C05459=1073.905,147.955,426.139,173.670,25.621,154.541
C05460=1073.899,147.705,426.161,173.668,25.618,154.541
C05461=1073.894,147.456,426.181,173.666,25.616,154.541
C05462=1073.888,147.208,426.202,173.664,25.613,154.541
C05463=1073.882,146.958,426.223,173.663,25.610,154.540
C05464=1073.877,146.709,426.244,173.661,25.608,154.540
C05465=1073.871,146.461,426.265,173.659,25.606,154.540
C05466=1073.865,146.211,426.286,173.657,25.603,154.539
C05467=1073.859,145.962,426.306,173.655,25.600,154.539
C05468=1073.854,145.714,426.327,173.654,25.598,154.539
C05469=1073.848,145.464,426.348,173.651,25.595,154.538
C05470=1073.843,145.215,426.369,173.650,25.592,154.538
C05471=1073.837,144.966,426.390,173.647,25.590,154.538
C05472=1073.830,144.717,426.410,173.646,25.587,154.537
C05473=1073.825,144.467,426.431,173.645,25.585,154.537
C05474=1073.820,144.219,426.452,173.642,25.582,154.537
C05475=1073.814,143.970,426.472,173.641,25.580,154.537
C05476=1073.808,143.720,426.493,173.638,25.577,154.536
C05477=1073.802,143.438,426.517,173.637,25.574,154.536
C05478=1073.795,143.157,426.540,173.635,25.571,154.535
C05479=1073.789,142.875,426.564,173.633,25.568,154.535
C05480=1073.782,142.593,426.586,173.630,25.565,154.535
C05481=1073.777,142.344,426.608,173.629,25.562,154.534
C05482=1073.771,142.094,426.628,173.626,25.560,154.534
C05483=1073.766,141.845,426.649,173.625,25.558,154.534
C05484=1073.760,141.596,426.669,173.624,25.555,154.533
C05485=1073.755,141.347,426.690,173.621,25.552,154.533
C05486=1073.748,141.098,426.711,173.620,25.550,154.533
C05487=1073.742,140.849,426.731,173.618,25.547,154.533
C05488=1073.737,140.600,426.752,173.616,25.544,154.532
C05489=1073.732,140.351,426.772,173.615,25.542,154.532
C05490=1073.727,140.102,426.793,173.612,25.539,154.532
C05491=1073.720,139.852,426.813,173.611,25.537,154.531
C05492=1073.715,139.603,426.834,173.609,25.534,154.531
C05493=1073.708,139.355,426.854,173.607,25.531,154.531
C05494=1073.703,139.106,426.875,173.606,25.529,154.530
C05495=1073.697,138.856,426.896,173.603,25.526,154.530
C05496=1073.691,138.607,426.916,173.602,25.523,154.530
C05497=1073.686,138.358,426.936,173.600,25.521,154.529
C05498=1073.680,138.109,426.956,173.598,25.518,154.529
C05499=1073.675,137.860,426.977,173.597,25.516,154.529
C05500=1073.668,137.611,426.997,173.595,25.513,154.528
C05501=1073.663,137.362,427.018,173.593,25.511,154.528
C05502=1073.658,137.112,427.038,173.591,25.508,154.528
C05503=1073.652,136.864,427.058,173.589,25.505,154.527
C05504=1073.647,136.615,427.079,173.588,25.503,154.527
C05505=1073.641,136.366,427.099,173.586,25.500,154.527
C05506=1073.635,136.116,427.120,173.584,25.497,154.527
C05507=1073.629,135.867,427.140,173.582,25.495,154.526
C05508=1073.623,135.618,427.160,173.580,25.493,154.526
C05509=1073.617,135.369,427.180,173.579,25.490,154.526
C05510=1073.612,135.120,427.201,173.577,25.487,154.525
C05511=1073.606,134.871,427.221,173.575,25.485,154.525
C05512=1073.600,134.621,427.242,173.574,25.482,154.525
C05513=1073.594,134.373,427.262,173.572,25.479,154.524
C05514=1073.589,134.123,427.282,173.570,25.477,154.524
C05515=1073.583,133.875,427.302,173.568,25.474,154.524
C05516=1073.578,133.625,427.322,173.566,25.472,154.523
C05517=1073.572,133.376,427.342,173.565,25.469,154.523
C05518=1073.567,133.127,427.362,173.563,25.466,154.523
C05519=1073.561,132.878,427.382,173.561,25.464,154.522
C05520=1073.555,132.628,427.403,173.560,25.461,154.522
C05521=1073.549,132.379,427.423,173.558,25.458,154.522
C05522=1073.544,132.130,427.444,173.556,25.456,154.522
C05523=1073.538,131.881,427.463,173.555,25.454,154.521
C05524=1073.532,131.632,427.483,173.552,25.450,154.521
C05525=1073.527,131.383,427.504,173.551,25.448,154.521
C05526=1073.521,131.134,427.523,173.549,25.446,154.520
C05527=1073.515,130.885,427.543,173.547,25.443,154.520
C05528=1073.509,130.635,427.563,173.546,25.440,154.520
C05529=1073.503,130.386,427.584,173.544,25.438,154.519
C05530=1073.497,130.137,427.604,173.542,25.435,154.519
C05531=1073.491,129.888,427.624,173.541,25.433,154.519
C05532=1073.486,129.639,427.643,173.538,25.430,154.518
C05533=1073.480,129.390,427.663,173.537,25.428,154.518
C05534=1073.474,129.141,427.683,173.535,25.425,154.518
C05535=1073.468,128.892,427.703,173.533,25.423,154.518
C05536=1073.462,128.642,427.723,173.532,25.420,154.517
C05537=1073.456,128.393,427.743,173.530,25.418,154.517
C05538=1073.451,128.144,427.763,173.528,25.415,154.517
C05539=1073.445,127.895,427.783,173.527,25.413,154.516
C05540=1073.439,127.646,427.803,173.525,25.410,154.516
C05541=1073.431,127.300,427.830,173.522,25.406,154.516
C05542=1073.423,126.955,427.858,173.520,25.403,154.515
C05543=1073.416,126.610,427.885,173.518,25.399,154.515
C05544=1073.407,126.264,427.912,173.516,25.396,154.514
C05545=1073.402,126.047,427.930,173.514,25.393,154.514
C05546=1073.398,125.829,427.947,173.513,25.391,154.514
C05547=1073.392,125.612,427.965,173.510,25.388,154.513
C05548=1073.387,125.394,427.981,173.509,25.386,154.513
C05549=1073.382,125.177,427.999,173.507,25.384,154.513
C05550=1073.377,124.959,428.017,173.506,25.382,154.513
C05551=1073.372,124.742,428.034,173.504,25.380,154.512
C05552=1073.367,124.524,428.051,173.503,25.377,154.512
C05553=1073.361,124.276,428.071,173.502,25.375,154.512
C05554=1073.355,124.026,428.090,173.500,25.372,154.511
C05555=1073.349,123.777,428.110,173.498,25.370,154.511
C05556=1073.344,123.528,428.130,173.497,25.367,154.511
C05557=1073.338,123.279,428.150,173.495,25.364,154.510
C05558=1073.333,123.029,428.169,173.493,25.362,154.510
C05559=1073.327,122.781,428.189,173.491,25.359,154.510
C05560=1073.321,122.531,428.208,173.490,25.357,154.509
C05561=1073.315,122.282,428.228,173.488,25.353,154.509
C05562=1073.310,122.033,428.248,173.486,25.351,154.509
C05563=1073.304,121.784,428.268,173.485,25.349,154.508
C05564=1073.298,121.534,428.287,173.484,25.346,154.508
C05565=1073.293,121.285,428.306,173.481,25.343,154.508
C05566=1073.287,121.037,428.326,173.480,25.341,154.508
C05567=1073.282,120.787,428.345,173.478,25.338,154.507
C05568=1073.276,120.538,428.365,173.476,25.336,154.507
C05569=1073.271,120.289,428.385,173.475,25.333,154.506
C05570=1073.265,120.039,428.404,173.473,25.330,154.506
C05571=1073.259,119.791,428.424,173.471,25.328,154.506
C05572=1073.253,119.541,428.444,173.470,25.325,154.506
C05573=1073.247,119.292,428.463,173.468,25.323,154.505
C05574=1073.242,119.043,428.483,173.467,25.320,154.505
C05575=1073.236,118.793,428.502,173.465,25.317,154.505
C05576=1073.230,118.545,428.522,173.463,25.314,154.504
C05577=1073.225,118.296,428.541,173.462,25.312,154.504
C05578=1073.220,118.046,428.561,173.459,25.309,154.504
C05579=1073.214,117.797,428.581,173.458,25.306,154.503
C05580=1073.208,117.548,428.600,173.457,25.304,154.503
C05581=1073.203,117.298,428.619,173.454,25.301,154.503
C05582=1073.197,117.050,428.639,173.453,25.299,154.502
C05583=1073.191,116.800,428.658,173.452,25.296,154.502
C05584=1073.185,116.551,428.678,173.450,25.293,154.502
C05585=1073.180,116.302,428.696,173.448,25.290,154.501
C05586=1073.174,116.053,428.716,173.447,25.288,154.501
C05587=1073.168,115.804,428.736,173.445,25.285,154.500
C05588=1073.163,115.554,428.755,173.443,25.282,154.500
C05589=1073.157,115.305,428.774,173.442,25.280,154.500
C05590=1073.152,115.057,428.794,173.440,25.277,154.500
C05591=1073.146,114.807,428.813,173.439,25.275,154.499
C05592=1073.141,114.558,428.833,173.437,25.272,154.499
C05593=1073.135,114.308,428.852,173.435,25.269,154.499
C05594=1073.129,114.059,428.871,173.434,25.267,154.498
C05595=1073.123,113.810,428.891,173.432,25.264,154.498
C05596=1073.117,113.561,428.910,173.430,25.261,154.497
C05597=1073.112,113.312,428.929,173.429,25.259,154.497
C05598=1073.107,113.063,428.948,173.427,25.256,154.497
C05599=1073.101,112.813,428.967,173.425,25.253,154.497
C05600=1073.095,112.564,428.986,173.424,25.251,154.496
C05601=1073.089,112.314,429.006,173.422,25.248,154.496
C05602=1073.083,112.065,429.024,173.421,25.246,154.496
C05603=1073.078,111.817,429.044,173.419,25.243,154.495
C05604=1073.072,111.568,429.063,173.417,25.240,154.495
C05605=1073.065,111.285,429.085,173.416,25.237,154.494
C05606=1073.058,111.003,429.107,173.414,25.235,154.494
C05607=1073.052,110.721,429.128,173.411,25.232,154.494
C05608=1073.045,110.439,429.149,173.410,25.229,154.493
C05609=1073.040,110.189,429.168,173.409,25.226,154.493
C05610=1073.035,109.940,429.187,173.406,25.223,154.493
C05611=1073.029,109.692,429.207,173.405,25.221,154.493
C05612=1073.022,109.442,429.226,173.404,25.219,154.492
C05613=1073.017,109.193,429.245,173.402,25.216,154.492
C05614=1073.011,108.944,429.264,173.400,25.213,154.492
C05615=1073.004,108.694,429.283,173.399,25.210,154.491
C05616=1073.000,108.445,429.301,173.397,25.208,154.491
C05617=1072.994,108.196,429.320,173.396,25.205,154.491
C05618=1072.988,107.947,429.339,173.394,25.202,154.490
C05619=1072.982,107.697,429.358,173.392,25.200,154.490
C05620=1072.977,107.448,429.377,173.391,25.197,154.489
C05621=1072.971,107.199,429.396,173.389,25.195,154.489
C05622=1072.965,106.950,429.415,173.387,25.192,154.489
C05623=1072.959,106.700,429.434,173.386,25.189,154.489
C05624=1072.953,106.451,429.453,173.384,25.187,154.488
C05625=1072.948,106.203,429.472,173.383,25.184,154.488
C05626=1072.942,105.953,429.491,173.381,25.181,154.488
C05627=1072.936,105.704,429.510,173.379,25.179,154.487
C05628=1072.930,105.455,429.528,173.378,25.176,154.487
C05629=1072.925,105.205,429.547,173.377,25.174,154.487
C05630=1072.919,104.956,429.566,173.374,25.171,154.486
C05631=1072.913,104.707,429.585,173.373,25.168,154.486
C05632=1072.908,104.458,429.604,173.372,25.166,154.486
C05633=1072.902,104.208,429.623,173.370,25.163,154.485
C05634=1072.896,103.959,429.642,173.368,25.160,154.485
C05635=1072.891,103.710,429.660,173.367,25.158,154.485
C05636=1072.885,103.461,429.679,173.365,25.155,154.484
C05637=1072.879,103.211,429.698,173.364,25.152,154.484
C05638=1072.873,102.962,429.717,173.361,25.150,154.484
C05639=1072.867,102.714,429.735,173.360,25.147,154.483
C05640=1072.862,102.464,429.754,173.359,25.145,154.483
C05641=1072.856,102.214,429.773,173.357,25.142,154.483
C05642=1072.850,101.966,429.791,173.356,25.139,154.482
C05643=1072.845,101.716,429.811,173.354,25.136,154.482
C05644=1072.839,101.466,429.829,173.352,25.134,154.482
C05645=1072.833,101.218,429.847,173.351,25.131,154.481
C05646=1072.828,100.968,429.867,173.350,25.129,154.481
C05647=1072.821,100.719,429.885,173.347,25.125,154.481
C05648=1072.817,100.470,429.903,173.346,25.123,154.480
C05649=1072.810,100.221,429.922,173.345,25.121,154.480
C05650=1072.804,99.971,429.941,173.343,25.118,154.480
C05651=1072.799,99.722,429.959,173.342,25.116,154.479
C05652=1072.792,99.473,429.977,173.340,25.113,154.479
C05653=1072.787,99.224,429.997,173.338,25.110,154.479
C05654=1072.781,98.975,430.014,173.337,25.108,154.478
C05655=1072.776,98.725,430.034,173.336,25.105,154.478
C05656=1072.769,98.476,430.052,173.333,25.102,154.478
C05657=1072.764,98.227,430.070,173.332,25.099,154.477
C05658=1072.758,97.978,430.089,173.331,25.097,154.477
C05659=1072.752,97.728,430.107,173.329,25.095,154.477
C05660=1072.747,97.479,430.126,173.328,25.092,154.476
C05661=1072.740,97.230,430.144,173.325,25.089,154.476
C05662=1072.734,96.980,430.162,173.324,25.086,154.476
C05663=1072.729,96.732,430.181,173.323,25.084,154.475
C05664=1072.723,96.482,430.199,173.321,25.081,154.475
C05665=1072.717,96.232,430.218,173.320,25.079,154.475
C05666=1072.712,95.983,430.236,173.318,25.076,154.474
C05667=1072.705,95.734,430.255,173.316,25.073,154.474
C05668=1072.701,95.485,430.273,173.315,25.071,154.474
C05669=1072.693,95.203,430.294,173.313,25.068,154.473
C05670=1072.687,94.921,430.315,173.312,25.065,154.473
C05671=1072.681,94.639,430.336,173.309,25.062,154.473
C05672=1072.674,94.356,430.356,173.308,25.059,154.472
C05673=1072.669,94.107,430.375,173.307,25.056,154.472
C05674=1072.662,93.858,430.393,173.305,25.054,154.471
C05675=1072.657,93.609,430.411,173.303,25.051,154.471
C05676=1072.651,93.360,430.430,173.302,25.048,154.471
C05677=1072.646,93.110,430.448,173.300,25.046,154.470
C05678=1072.639,92.861,430.466,173.299,25.043,154.470
C05679=1072.634,92.611,430.485,173.298,25.040,154.470
C05680=1072.628,92.363,430.503,173.295,25.037,154.469
C05681=1072.622,92.113,430.521,173.294,25.035,154.469
C05682=1072.617,91.864,430.539,173.293,25.032,154.469
C05683=1072.611,91.615,430.558,173.291,25.030,154.468
C05684=1072.605,91.366,430.575,173.290,25.027,154.468
C05685=1072.599,91.116,430.595,173.288,25.024,154.468
C05686=1072.594,90.867,430.612,173.286,25.021,154.467
C05687=1072.588,90.617,430.630,173.285,25.019,154.467
C05688=1072.582,90.369,430.648,173.284,25.016,154.467
C05689=1072.577,90.119,430.667,173.282,25.014,154.466
C05690=1072.570,89.869,430.685,173.280,25.010,154.466
C05691=1072.565,89.621,430.703,173.279,25.008,154.466
C05692=1072.559,89.371,430.721,173.277,25.006,154.465
C05693=1072.553,89.122,430.739,173.276,25.003,154.465
C05694=1072.547,88.873,430.757,173.275,25.001,154.465
C05695=1072.541,88.624,430.775,173.272,24.997,154.464
C05696=1072.535,88.374,430.793,173.271,24.995,154.464
C05697=1072.530,88.125,430.811,173.270,24.993,154.464
C05698=1072.524,87.876,430.830,173.268,24.990,154.463
C05699=1072.518,87.627,430.847,173.267,24.987,154.463
C05700=1072.512,87.377,430.865,173.266,24.985,154.463
C05701=1072.507,87.128,430.883,173.263,24.982,154.462
C05702=1072.500,86.879,430.901,173.262,24.979,154.462
C05703=1072.495,86.630,430.919,173.261,24.977,154.462
C05704=1072.489,86.380,430.937,173.259,24.974,154.461
C05705=1072.483,86.131,430.954,173.258,24.971,154.461
C05706=1072.477,85.881,430.972,173.256,24.969,154.461
C05707=1072.472,85.632,430.991,173.254,24.966,154.460
C05708=1072.466,85.383,431.009,173.253,24.964,154.460
C05709=1072.460,85.134,431.027,173.252,24.961,154.460
C05710=1072.454,84.884,431.045,173.250,24.958,154.459
C05711=1072.448,84.635,431.062,173.249,24.955,154.459
C05712=1072.442,84.386,431.081,173.247,24.953,154.459
C05713=1072.437,84.137,431.098,173.245,24.950,154.458
C05714=1072.430,83.887,431.116,173.244,24.948,154.458
C05715=1072.425,83.638,431.134,173.243,24.945,154.458
C05716=1072.419,83.388,431.152,173.241,24.942,154.457
C05717=1072.413,83.139,431.169,173.240,24.939,154.457
C05718=1072.408,82.890,431.187,173.238,24.937,154.457
C05719=1072.402,82.640,431.205,173.236,24.934,154.456
C05720=1072.396,82.391,431.222,173.235,24.932,154.456
C05721=1072.390,82.142,431.240,173.234,24.929,154.456
C05722=1072.385,81.893,431.259,173.232,24.926,154.455
C05723=1072.379,81.643,431.277,173.231,24.923,154.455
C05724=1072.373,81.394,431.295,173.229,24.921,154.455
C05725=1072.368,81.145,431.312,173.227,24.918,154.454
C05726=1072.362,80.895,431.330,173.226,24.916,154.454
C05727=1072.356,80.646,431.348,173.225,24.913,154.454
C05728=1072.350,80.396,431.366,173.223,24.910,154.453
C05729=1072.344,80.147,431.383,173.222,24.907,154.453
C05730=1072.339,79.898,431.401,173.220,24.905,154.453
C05731=1072.333,79.649,431.419,173.218,24.902,154.452
C05732=1072.327,79.400,431.436,173.217,24.900,154.452
C05733=1072.321,79.117,431.456,173.216,24.897,154.452
C05734=1072.314,78.835,431.476,173.214,24.893,154.451
C05735=1072.307,78.554,431.496,173.212,24.891,154.451
C05736=1072.301,78.271,431.516,173.210,24.887,154.450
C05737=1072.295,78.022,431.533,173.209,24.884,154.450
C05738=1072.289,77.773,431.551,173.207,24.882,154.450
C05739=1072.284,77.524,431.569,173.206,24.879,154.449
C05740=1072.278,77.274,431.586,173.205,24.877,154.449
C05741=1072.271,77.025,431.604,173.203,24.874,154.449
C05742=1072.266,76.776,431.621,173.201,24.871,154.448
C05743=1072.260,76.526,431.639,173.200,24.868,154.448
C05744=1072.255,76.277,431.656,173.198,24.866,154.448
C05745=1072.249,76.028,431.674,173.197,24.863,154.447
C05746=1072.242,75.778,431.691,173.196,24.861,154.447
C05747=1072.237,75.529,431.709,173.194,24.858,154.447
C05748=1072.231,75.280,431.726,173.193,24.856,154.446
C05749=1072.225,75.030,431.744,173.191,24.853,154.446
C05750=1072.220,74.781,431.761,173.190,24.850,154.446
C05751=1072.214,74.532,431.778,173.188,24.848,154.445
C05752=1072.207,74.282,431.796,173.187,24.845,154.445
C05753=1072.202,74.033,431.813,173.185,24.842,154.445
C05754=1072.196,73.784,431.831,173.184,24.840,154.444
C05755=1072.191,73.534,431.848,173.183,24.837,154.444
C05756=1072.184,73.285,431.865,173.181,24.834,154.444
C05757=1072.179,73.036,431.883,173.179,24.832,154.443
C05758=1072.173,72.786,431.901,173.178,24.829,154.443
C05759=1072.167,72.537,431.918,173.177,24.826,154.443
C05760=1072.161,72.288,431.935,173.175,24.823,154.442
C05761=1072.155,72.038,431.952,173.174,24.821,154.442
C05762=1072.150,71.789,431.970,173.173,24.818,154.441
C05763=1072.144,71.539,431.987,173.170,24.816,154.441
C05764=1072.138,71.291,432.004,173.169,24.813,154.441
C05765=1072.132,71.041,432.022,173.168,24.810,154.441
C05766=1072.126,70.792,432.039,173.166,24.807,154.440
C05767=1072.121,70.542,432.056,173.165,24.805,154.440
C05768=1072.114,70.293,432.074,173.164,24.802,154.439
C05769=1072.109,70.044,432.091,173.162,24.800,154.439
C05770=1072.104,69.794,432.108,173.160,24.797,154.439
C05771=1072.097,69.545,432.125,173.159,24.794,154.439
C05772=1072.091,69.296,432.143,173.157,24.791,154.438
C05773=1072.086,69.046,432.160,173.156,24.789,154.438
C05774=1072.080,68.797,432.177,173.155,24.786,154.437
C05775=1072.075,68.548,432.194,173.153,24.784,154.437
C05776=1072.068,68.298,432.211,173.152,24.781,154.437
C05777=1072.062,68.049,432.228,173.150,24.778,154.436
C05778=1072.057,67.799,432.245,173.149,24.775,154.436
C05779=1072.051,67.551,432.262,173.147,24.773,154.436
C05780=1072.045,67.300,432.279,173.146,24.770,154.435
C05781=1072.039,67.052,432.296,173.145,24.768,154.435
C05782=1072.033,66.803,432.314,173.143,24.765,154.435
C05783=1072.028,66.553,432.331,173.142,24.762,154.434
C05784=1072.021,66.304,432.348,173.141,24.759,154.434
C05785=1072.016,66.054,432.365,173.138,24.757,154.434
C05786=1072.010,65.805,432.382,173.137,24.754,154.433
C05787=1072.004,65.555,432.399,173.136,24.752,154.433
C05788=1071.998,65.306,432.416,173.134,24.749,154.433
C05789=1071.992,65.056,432.433,173.133,24.746,154.432
C05790=1071.986,64.808,432.450,173.132,24.743,154.432
C05791=1071.981,64.558,432.467,173.130,24.741,154.432
C05792=1071.975,64.309,432.484,173.129,24.738,154.431
C05793=1071.969,64.059,432.501,173.127,24.735,154.431
C05794=1071.963,63.810,432.518,173.125,24.733,154.431
C05795=1071.957,63.561,432.534,173.124,24.730,154.430
C05796=1071.950,63.311,432.552,173.123,24.728,154.430
C05797=1071.944,63.029,432.570,173.121,24.725,154.430
C05798=1071.938,62.747,432.590,173.119,24.722,154.429
C05799=1071.930,62.465,432.609,173.118,24.719,154.429
C05800=1071.924,62.182,432.628,173.116,24.716,154.428
C05801=1071.918,61.934,432.645,173.115,24.713,154.428
C05802=1071.912,61.684,432.661,173.113,24.711,154.428
C05803=1071.906,61.434,432.678,173.112,24.708,154.428
C05804=1071.900,61.185,432.695,173.110,24.706,154.427
C05805=1071.894,60.936,432.712,173.109,24.703,154.427
C05806=1071.888,60.687,432.729,173.108,24.700,154.427
C05807=1071.882,60.437,432.745,173.106,24.698,154.426
C05808=1071.876,60.187,432.762,173.104,24.695,154.426
C05809=1071.870,59.939,432.779,173.103,24.692,154.426
C05810=1071.864,59.689,432.796,173.102,24.689,154.425
C05811=1071.858,59.440,432.812,173.100,24.687,154.425
C05812=1071.852,59.191,432.829,173.099,24.684,154.425
C05813=1071.846,58.940,432.846,173.098,24.682,154.424
C05814=1071.840,58.691,432.863,173.096,24.679,154.424
C05815=1071.834,58.442,432.879,173.095,24.677,154.424
C05816=1071.828,58.193,432.896,173.093,24.674,154.423
C05817=1071.823,57.943,432.913,173.091,24.671,154.423
C05818=1071.817,57.694,432.929,173.090,24.669,154.423
C05819=1071.811,57.445,432.945,173.089,24.666,154.422
C05820=1071.805,57.195,432.963,173.087,24.663,154.422
C05821=1071.799,56.946,432.979,173.086,24.660,154.422
C05822=1071.793,56.696,432.996,173.085,24.658,154.421
C05823=1071.787,56.447,433.012,173.083,24.655,154.421
C05824=1071.782,56.198,433.030,173.082,24.653,154.421
C05825=1071.776,55.949,433.046,173.080,24.650,154.420
C05826=1071.770,55.699,433.062,173.079,24.647,154.420
C05827=1071.764,55.450,433.078,173.077,24.645,154.420
C05828=1071.759,55.200,433.095,173.076,24.642,154.419
C05829=1071.752,54.951,433.112,173.075,24.640,154.419
C05830=1071.746,54.701,433.129,173.073,24.637,154.419
C05831=1071.740,54.452,433.145,173.072,24.634,154.418
C05832=1071.735,54.202,433.162,173.071,24.631,154.418
C05833=1071.729,53.953,433.178,173.069,24.629,154.418
C05834=1071.723,53.704,433.194,173.067,24.626,154.417
C05835=1071.716,53.455,433.211,173.066,24.623,154.417
C05836=1071.711,53.205,433.228,173.064,24.621,154.416
C05837=1071.705,52.956,433.244,173.063,24.618,154.416
C05838=1071.699,52.707,433.261,173.062,24.615,154.416
C05839=1071.693,52.457,433.277,173.060,24.613,154.416
C05840=1071.688,52.208,433.294,173.059,24.610,154.415
C05841=1071.682,51.958,433.310,173.058,24.608,154.415
C05842=1071.676,51.709,433.326,173.057,24.605,154.414
C05843=1071.670,51.460,433.343,173.055,24.602,154.414
C05844=1071.664,51.210,433.359,173.053,24.599,154.414
C05845=1071.659,50.961,433.376,173.052,24.597,154.413
C05846=1071.653,50.711,433.392,173.050,24.594,154.413
C05847=1071.647,50.462,433.408,173.049,24.591,154.413
C05848=1071.641,50.212,433.424,173.048,24.589,154.412
C05849=1071.635,49.964,433.441,173.046,24.586,154.412
C05850=1071.630,49.714,433.458,173.045,24.583,154.412
C05851=1071.624,49.465,433.475,173.044,24.581,154.411
C05852=1071.618,49.215,433.491,173.043,24.578,154.411
C05853=1071.612,48.966,433.507,173.041,24.576,154.411
C05854=1071.606,48.716,433.523,173.039,24.572,154.410
C05855=1071.601,48.466,433.539,173.038,24.570,154.410
C05856=1071.595,48.217,433.556,173.036,24.567,154.410
C05857=1071.589,47.968,433.572,173.035,24.565,154.409
C05858=1071.583,47.718,433.588,173.034,24.562,154.409
C05859=1071.577,47.469,433.604,173.032,24.559,154.409
C05860=1071.571,47.220,433.621,173.031,24.557,154.408
C05861=1071.565,46.937,433.640,173.029,24.553,154.408
C05862=1071.559,46.655,433.658,173.028,24.550,154.408
C05863=1071.552,46.372,433.676,173.027,24.547,154.407
C05864=1071.546,46.090,433.695,173.024,24.544,154.407
C05865=1071.540,45.840,433.711,173.023,24.541,154.406
C05866=1071.534,45.591,433.728,173.022,24.539,154.406
C05867=1071.528,45.342,433.743,173.021,24.536,154.406
C05868=1071.522,45.093,433.760,173.019,24.534,154.405
C05869=1071.517,44.843,433.775,173.018,24.531,154.405
C05870=1071.511,44.594,433.791,173.017,24.528,154.405
C05871=1071.506,44.344,433.808,173.015,24.525,154.404
C05872=1071.500,44.095,433.825,173.014,24.523,154.404
C05873=1071.494,43.845,433.841,173.012,24.520,154.404
C05874=1071.488,43.596,433.857,173.010,24.517,154.403
C05875=1071.482,43.346,433.873,173.009,24.515,154.403
C05876=1071.476,43.097,433.889,173.008,24.512,154.403
C05877=1071.470,42.847,433.905,173.007,24.509,154.402
C05878=1071.465,42.599,433.921,173.005,24.507,154.402
C05879=1071.458,42.350,433.937,173.004,24.504,154.402
C05880=1071.452,42.100,433.952,173.003,24.502,154.401
C05881=1071.447,41.850,433.969,173.001,24.499,154.401
C05882=1071.441,41.601,433.985,173.000,24.496,154.401
C05883=1071.435,41.352,434.001,172.999,24.493,154.400
C05884=1071.429,41.102,434.017,172.996,24.491,154.400
C05885=1071.423,40.852,434.033,172.995,24.488,154.400
C05886=1071.417,40.603,434.049,172.994,24.485,154.399
C05887=1071.411,40.353,434.065,172.992,24.483,154.399
C05888=1071.405,40.104,434.081,172.991,24.480,154.399
C05889=1071.400,39.855,434.097,172.990,24.478,154.398
C05890=1071.394,39.606,434.113,172.989,24.475,154.398
C05891=1071.389,39.356,434.129,172.987,24.472,154.398
C05892=1071.382,39.107,434.144,172.986,24.470,154.397
C05893=1071.376,38.857,434.160,172.985,24.467,154.397
C05894=1071.370,38.607,434.176,172.983,24.464,154.397
C05895=1071.364,38.358,434.192,172.982,24.462,154.396
C05896=1071.359,38.109,434.207,172.980,24.459,154.396
C05897=1071.353,37.859,434.224,172.978,24.456,154.396
C05898=1071.347,37.610,434.240,172.977,24.453,154.395
C05899=1071.341,37.360,434.255,172.976,24.451,154.395
C05900=1071.335,37.111,434.271,172.974,24.449,154.395
C05901=1071.329,36.862,434.287,172.973,24.446,154.394
C05902=1071.323,36.612,434.303,172.972,24.443,154.394
C05903=1071.317,36.363,434.319,172.971,24.440,154.394
C05904=1071.312,36.113,434.334,172.969,24.438,154.393
C05905=1071.306,35.864,434.350,172.968,24.436,154.393
C05906=1071.299,35.614,434.365,172.967,24.433,154.393
C05907=1071.293,35.365,434.381,172.964,24.430,154.392
C05908=1071.287,35.116,434.398,172.963,24.427,154.392
C05909=1071.282,34.866,434.413,172.962,24.425,154.392
C05910=1071.276,34.617,434.428,172.960,24.422,154.391
C05911=1071.270,34.367,434.444,172.959,24.419,154.391
C05912=1071.264,34.118,434.460,172.958,24.417,154.391
C05913=1071.258,33.868,434.475,172.957,24.414,154.390
C05914=1071.252,33.619,434.491,172.955,24.412,154.390
C05915=1071.246,33.369,434.507,172.954,24.409,154.390
C05916=1071.240,33.121,434.522,172.953,24.406,154.389
C05917=1071.234,32.871,434.538,172.951,24.404,154.389
C05918=1071.228,32.621,434.554,172.950,24.401,154.389
C05919=1071.223,32.371,434.570,172.948,24.398,154.388
C05920=1071.216,32.122,434.584,172.946,24.396,154.388
C05921=1071.211,31.873,434.600,172.945,24.393,154.388
C05922=1071.205,31.623,434.616,172.944,24.391,154.387
C05923=1071.199,31.374,434.632,172.943,24.388,154.387
C05924=1071.193,31.124,434.647,172.941,24.385,154.387
C05925=1071.187,30.842,434.665,172.940,24.382,154.386
C05926=1071.179,30.559,434.682,172.938,24.379,154.386
C05927=1071.173,30.277,434.699,172.937,24.376,154.386
C05928=1071.167,29.995,434.717,172.935,24.373,154.385
C05929=1071.161,29.746,434.732,172.934,24.371,154.385
C05930=1071.155,29.496,434.749,172.932,24.368,154.385
C05931=1071.149,29.246,434.764,172.931,24.365,154.384
C05932=1071.143,28.997,434.779,172.929,24.363,154.384
C05933=1071.137,28.748,434.795,172.928,24.360,154.384
C05934=1071.132,28.498,434.811,172.927,24.358,154.383
C05935=1071.125,28.248,434.826,172.925,24.355,154.383
C05936=1071.120,28.000,434.841,172.924,24.352,154.383
C05937=1071.114,27.750,434.856,172.923,24.350,154.382
C05938=1071.108,27.500,434.872,172.921,24.348,154.382
C05939=1071.101,27.250,434.887,172.920,24.345,154.382
C05940=1071.096,27.002,434.903,172.919,24.342,154.381
C05941=1071.090,26.752,434.918,172.917,24.339,154.381
C05942=1071.084,26.502,434.933,172.916,24.337,154.381
C05943=1071.077,26.253,434.949,172.914,24.334,154.380
C05944=1071.072,26.004,434.964,172.913,24.331,154.380
C05945=1071.066,25.754,434.979,172.911,24.329,154.380
C05946=1071.060,25.504,434.995,172.910,24.327,154.379
C05947=1071.054,25.255,435.010,172.909,24.324,154.379
C05948=1071.048,25.006,435.025,172.907,24.321,154.379
C05949=1071.042,24.756,435.040,172.906,24.319,154.378
C05950=1071.036,24.507,435.055,172.905,24.316,154.378
C05951=1071.031,24.257,435.070,172.903,24.314,154.378
C05952=1071.024,24.008,435.086,172.902,24.311,154.377
C05953=1071.018,23.758,435.102,172.901,24.308,154.377
C05954=1071.013,23.509,435.116,172.899,24.306,154.377
C05955=1071.007,23.259,435.132,172.898,24.303,154.377
C05956=1071.001,23.010,435.147,172.897,24.301,154.376
C05957=1070.995,22.761,435.161,172.894,24.298,154.376
C05958=1070.989,22.511,435.178,172.893,24.295,154.376
C05959=1070.983,22.262,435.193,172.892,24.292,154.375
C05960=1070.977,22.012,435.208,172.891,24.290,154.375
C05961=1070.971,21.763,435.223,172.889,24.287,154.375
C05962=1070.965,21.513,435.238,172.888,24.285,154.374
C05963=1070.960,21.264,435.253,172.887,24.282,154.374
C05964=1070.953,21.014,435.268,172.885,24.279,154.374
C05965=1070.948,20.764,435.283,172.884,24.277,154.373
C05966=1070.942,20.515,435.298,172.883,24.275,154.373
C05967=1070.936,20.265,435.313,172.881,24.272,154.373
C05968=1070.930,20.016,435.329,172.880,24.269,154.372
C05969=1070.924,19.767,435.344,172.879,24.267,154.372
C05970=1070.918,19.517,435.359,172.877,24.264,154.372
C05971=1070.912,19.268,435.374,172.875,24.261,154.371
C05972=1070.906,19.019,435.389,172.874,24.259,154.371
C05973=1070.900,18.769,435.404,172.873,24.257,154.371
C05974=1070.894,18.519,435.419,172.871,24.254,154.370
C05975=1070.888,18.270,435.434,172.870,24.251,154.370
C05976=1070.882,18.020,435.449,172.869,24.249,154.370
C05977=1070.877,17.771,435.464,172.867,24.246,154.369
C05978=1070.870,17.522,435.479,172.866,24.244,154.369
C05979=1070.864,17.272,435.494,172.865,24.241,154.369
C05980=1070.858,17.023,435.508,172.863,24.238,154.368
C05981=1070.853,16.773,435.524,172.862,24.236,154.368
C05982=1070.847,16.524,435.538,172.861,24.233,154.368
C05983=1070.840,16.274,435.553,172.860,24.231,154.368
C05984=1070.835,16.024,435.569,172.857,24.228,154.367
C05985=1070.829,15.775,435.583,172.856,24.225,154.367
C05986=1070.823,15.525,435.598,172.855,24.223,154.367
C05987=1070.817,15.276,435.612,172.853,24.220,154.366
C05988=1070.811,15.026,435.628,172.852,24.218,154.366
C05989=1070.804,14.746,435.644,172.851,24.215,154.366
C05990=1070.798,14.465,435.661,172.850,24.212,154.365
C05991=1070.792,14.184,435.678,172.847,24.209,154.365
C05992=1070.784,13.902,435.695,172.846,24.206,154.365
C05993=1070.778,13.653,435.709,172.845,24.204,154.364
C05994=1070.772,13.403,435.725,172.843,24.201,154.364
C05995=1070.767,13.154,435.739,172.842,24.199,154.364
C05996=1070.760,12.904,435.753,172.841,24.196,154.363
C05997=1070.754,12.655,435.768,172.839,24.194,154.363
C05998=1070.748,12.406,435.783,172.837,24.191,154.363
C05999=1070.742,12.156,435.798,172.836,24.189,154.363
C06000=1070.736,11.907,435.813,172.834,24.186,154.362
C06001=1070.730,11.657,435.827,172.833,24.184,154.362
C06002=1070.724,11.407,435.842,172.832,24.181,154.362
C06003=1070.718,11.158,435.856,172.831,24.178,154.361
C06004=1070.711,10.908,435.871,172.829,24.176,154.361
C06005=1070.706,10.659,435.886,172.828,24.174,154.361
C06006=1070.700,10.409,435.900,172.826,24.171,154.360
C06007=1070.694,10.160,435.915,172.825,24.168,154.360
C06008=1070.687,9.911,435.930,172.824,24.166,154.360
C06009=1070.682,9.662,435.944,172.823,24.164,154.360
C06010=1070.676,9.411,435.958,172.821,24.161,154.359
C06011=1070.670,9.162,435.973,172.820,24.159,154.359
C06012=1070.663,8.913,435.988,172.818,24.155,154.359
C06013=1070.658,8.663,436.002,172.816,24.153,154.358
C06014=1070.652,8.413,436.017,172.815,24.151,154.358
C06015=1070.645,8.164,436.032,172.814,24.148,154.358
C06016=1070.639,7.915,436.046,172.812,24.146,154.357
C06017=1070.633,7.665,436.060,172.811,24.143,154.357
C06018=1070.627,7.416,436.075,172.810,24.141,154.357
C06019=1070.621,7.166,436.090,172.808,24.138,154.357
C06020=1070.616,6.916,436.104,172.807,24.136,154.356
C06021=1070.610,6.667,436.118,172.806,24.133,154.356
C06022=1070.604,6.417,436.133,172.804,24.130,154.356
C06023=1070.598,6.168,436.147,172.803,24.128,154.355
C06024=1070.592,5.919,436.162,172.802,24.126,154.355
C06025=1070.586,5.669,436.176,172.800,24.123,154.355
C06026=1070.580,5.419,436.191,172.798,24.121,154.354
C06027=1070.574,5.170,436.206,172.797,24.118,154.354
C06028=1070.568,4.920,436.220,172.796,24.115,154.354
C06029=1070.562,4.671,436.234,172.794,24.113,154.354
C06030=1070.556,4.421,436.249,172.793,24.110,154.353
C06031=1070.550,4.172,436.263,172.792,24.108,154.353
C06032=1070.545,3.922,436.277,172.790,24.105,154.353
C06033=1070.538,3.673,436.292,172.789,24.103,154.352
C06034=1070.533,3.424,436.307,172.788,24.100,154.352
C06035=1070.527,3.173,436.321,172.786,24.098,154.352
C06036=1070.521,2.925,436.335,172.785,24.096,154.351
C06037=1070.515,2.674,436.350,172.784,24.093,154.351
C06038=1070.509,2.425,436.364,172.782,24.090,154.351
C06039=1070.503,2.176,436.378,172.781,24.088,154.350
C06040=1070.497,1.926,436.393,172.780,24.085,154.350
C06041=1070.492,1.676,436.407,172.777,24.083,154.350
C06042=1070.485,1.427,436.422,172.776,24.080,154.350
C06043=1070.480,1.177,436.436,172.775,24.077,154.349
C06044=1070.474,0.928,436.450,172.774,24.075,154.349
C06045=1070.467,0.678,436.464,172.772,24.073,154.349
C06046=1070.461,0.429,436.479,172.771,24.070,154.348
C06047=1070.456,0.180,436.492,172.770,24.068,154.348
C06048=1070.450,-0.070,436.507,172.768,24.065,154.348
C06049=1070.444,-0.319,436.521,172.767,24.062,154.348
C06050=1070.439,-0.569,436.535,172.766,24.060,154.347
C06051=1070.432,-0.819,436.550,172.764,24.058,154.347
C06052=1070.427,-1.068,436.564,172.763,24.055,154.347
C06053=1070.420,-1.348,436.580,172.761,24.052,154.346
C06054=1070.413,-1.626,436.596,172.759,24.050,154.346
C06055=1070.407,-1.905,436.612,172.758,24.047,154.346
C06056=1070.400,-2.185,436.628,172.756,24.044,154.345
C06057=1070.394,-2.434,436.642,172.755,24.041,154.345
C06058=1070.389,-2.683,436.656,172.753,24.038,154.345
C06059=1070.382,-2.933,436.670,172.752,24.036,154.344
C06060=1070.376,-3.182,436.684,172.751,24.034,154.344
C06061=1070.371,-3.432,436.698,172.749,24.031,154.344
C06062=1070.365,-3.682,436.712,172.748,24.029,154.344
C06063=1070.358,-3.931,436.726,172.747,24.026,154.343
C06064=1070.353,-4.180,436.740,172.745,24.024,154.343
C06065=1070.347,-4.431,436.754,172.744,24.022,154.343
C06066=1070.340,-4.679,436.768,172.743,24.019,154.343
C06067=1070.335,-4.929,436.782,172.741,24.017,154.342
C06068=1070.329,-5.179,436.797,172.740,24.015,154.342
C06069=1070.322,-5.429,436.810,172.739,24.012,154.342
C06070=1070.316,-5.678,436.825,172.736,24.009,154.341
C06071=1070.311,-5.928,436.839,172.735,24.006,154.341
C06072=1070.304,-6.177,436.852,172.734,24.004,154.341
C06073=1070.298,-6.427,436.866,172.733,24.002,154.340
C06074=1070.292,-6.676,436.880,172.731,23.999,154.340
C06075=1070.286,-6.926,436.894,172.730,23.997,154.340
C06076=1070.281,-7.175,436.908,172.729,23.994,154.340
C06077=1070.274,-7.425,436.921,172.727,23.992,154.339
C06078=1070.268,-7.674,436.936,172.726,23.990,154.339
C06079=1070.263,-7.924,436.950,172.724,23.987,154.339
C06080=1070.256,-8.174,436.964,172.723,23.985,154.339
C06081=1070.251,-8.423,436.977,172.722,23.982,154.338
C06082=1070.244,-8.672,436.991,172.720,23.980,154.338
C06083=1070.238,-8.923,437.005,172.719,23.978,154.338
C06084=1070.232,-9.172,437.019,172.717,23.975,154.337
C06085=1070.226,-9.421,437.033,172.716,23.972,154.337
C06086=1070.221,-9.670,437.047,172.714,23.970,154.337
C06087=1070.214,-9.920,437.060,172.713,23.968,154.337
C06088=1070.208,-10.170,437.074,172.711,23.965,154.336
C06089=1070.203,-10.420,437.088,172.710,23.963,154.336
C06090=1070.197,-10.669,437.101,172.709,23.960,154.336
C06091=1070.191,-10.919,437.115,172.707,23.958,154.336
C06092=1070.184,-11.168,437.129,172.706,23.956,154.335
C06093=1070.179,-11.417,437.143,172.705,23.953,154.335
C06094=1070.172,-11.667,437.157,172.703,23.951,154.335
C06095=1070.166,-11.917,437.171,172.702,23.948,154.334
C06096=1070.161,-12.166,437.185,172.701,23.946,154.334
C06097=1070.155,-12.416,437.198,172.699,23.944,154.334
C06098=1070.149,-12.665,437.212,172.698,23.941,154.334
C06099=1070.143,-12.915,437.225,172.696,23.938,154.333
C06100=1070.137,-13.165,437.239,172.694,23.936,154.333
C06101=1070.131,-13.414,437.253,172.693,23.934,154.333
C06102=1070.125,-13.664,437.266,172.692,23.931,154.333
C06103=1070.120,-13.913,437.280,172.690,23.929,154.332
C06104=1070.114,-14.163,437.294,172.689,23.926,154.332
C06105=1070.107,-14.413,437.308,172.688,23.924,154.332
C06106=1070.101,-14.662,437.321,172.686,23.922,154.331
C06107=1070.096,-14.912,437.335,172.685,23.920,154.331
C06108=1070.090,-15.161,437.348,172.684,23.917,154.331
C06109=1070.084,-15.410,437.362,172.682,23.915,154.331
C06110=1070.077,-15.660,437.376,172.681,23.913,154.330
C06111=1070.071,-15.910,437.389,172.680,23.910,154.330
C06112=1070.066,-16.159,437.403,172.678,23.908,154.330
C06113=1070.059,-16.409,437.416,172.676,23.905,154.330
C06114=1070.053,-16.658,437.429,172.675,23.903,154.329
C06115=1070.047,-16.908,437.444,172.673,23.901,154.329
C06116=1070.041,-17.157,437.457,172.672,23.898,154.329
C06117=1070.035,-17.435,437.472,172.671,23.896,154.329
C06118=1070.027,-17.712,437.487,172.669,23.893,154.328
C06119=1070.021,-17.990,437.502,172.667,23.890,154.328
C06120=1070.014,-18.268,437.516,172.666,23.888,154.328
C06121=1070.009,-18.517,437.530,172.664,23.885,154.328
C06122=1070.002,-18.766,437.543,172.663,23.883,154.327
C06123=1069.996,-19.016,437.557,172.662,23.881,154.327
C06124=1069.990,-19.266,437.571,172.660,23.879,154.327
C06125=1069.984,-19.515,437.584,172.659,23.876,154.327
C06126=1069.978,-19.765,437.597,172.658,23.874,154.326
C06127=1069.972,-20.014,437.610,172.656,23.872,154.326
C06128=1069.966,-20.264,437.624,172.654,23.869,154.326
C06129=1069.960,-20.513,437.637,172.653,23.866,154.325
C06130=1069.954,-20.762,437.650,172.651,23.865,154.325
C06131=1069.948,-21.012,437.664,172.650,23.862,154.325
C06132=1069.942,-21.263,437.677,172.648,23.860,154.325
C06133=1069.936,-21.512,437.690,172.647,23.857,154.324
C06134=1069.930,-21.761,437.704,172.646,23.855,154.324
C06135=1069.924,-22.011,437.717,172.644,23.853,154.324
C06136=1069.918,-22.261,437.730,172.643,23.851,154.324
C06137=1069.913,-22.510,437.744,172.642,23.848,154.324
C06138=1069.906,-22.759,437.757,172.640,23.846,154.323
C06139=1069.900,-23.009,437.770,172.639,23.843,154.323
C06140=1069.894,-23.259,437.783,172.638,23.841,154.323
C06141=1069.889,-23.508,437.797,172.636,23.839,154.323
C06142=1069.882,-23.758,437.810,172.634,23.836,154.322
C06143=1069.876,-24.008,437.823,172.633,23.834,154.322
C06144=1069.870,-24.257,437.836,172.631,23.832,154.322
C06145=1069.864,-24.507,437.850,172.630,23.829,154.321
C06146=1069.858,-24.756,437.863,172.628,23.827,154.321
C06147=1069.852,-25.006,437.876,172.627,23.825,154.321
C06148=1069.847,-25.256,437.890,172.626,23.823,154.321
C06149=1069.841,-25.505,437.903,172.624,23.820,154.321
C06150=1069.835,-25.755,437.916,172.623,23.818,154.320
C06151=1069.828,-26.004,437.929,172.622,23.816,154.320
C06152=1069.823,-26.254,437.943,172.620,23.813,154.320
C06153=1069.817,-26.503,437.955,172.619,23.811,154.320
C06154=1069.811,-26.753,437.969,172.618,23.809,154.319
C06155=1069.805,-27.003,437.981,172.616,23.807,154.319
C06156=1069.799,-27.252,437.994,172.615,23.804,154.319
C06157=1069.792,-27.501,438.008,172.613,23.802,154.319
C06158=1069.787,-27.751,438.020,172.611,23.800,154.318
C06159=1069.780,-28.000,438.034,172.610,23.797,154.318
C06160=1069.774,-28.251,438.046,172.608,23.795,154.318
C06161=1069.768,-28.500,438.060,172.607,23.793,154.318
C06162=1069.762,-28.750,438.073,172.606,23.791,154.317
C06163=1069.756,-29.000,438.086,172.604,23.788,154.317
C06164=1069.750,-29.249,438.099,172.603,23.786,154.317
C06165=1069.744,-29.499,438.112,172.601,23.784,154.317
C06166=1069.738,-29.748,438.125,172.600,23.782,154.317
C06167=1069.732,-29.998,438.138,172.599,23.780,154.316
C06168=1069.726,-30.247,438.151,172.597,23.777,154.316
C06169=1069.720,-30.497,438.164,172.596,23.775,154.316
C06170=1069.714,-30.746,438.177,172.594,23.773,154.316
C06171=1069.708,-30.996,438.189,172.592,23.770,154.315
C06172=1069.702,-31.245,438.203,172.591,23.768,154.315
C06173=1069.696,-31.495,438.215,172.589,23.766,154.315
C06174=1069.689,-31.745,438.229,172.588,23.764,154.315
C06175=1069.684,-31.994,438.241,172.587,23.762,154.315
C06176=1069.678,-32.244,438.254,172.585,23.759,154.314
C06177=1069.671,-32.494,438.267,172.584,23.757,154.314
C06178=1069.665,-32.743,438.279,172.582,23.755,154.314
C06179=1069.659,-32.993,438.293,172.581,23.753,154.314
C06180=1069.653,-33.243,438.305,172.580,23.751,154.313
C06181=1069.647,-33.519,438.320,172.578,23.748,154.313
C06182=1069.640,-33.796,438.334,172.576,23.746,154.313
C06183=1069.634,-34.072,438.348,172.575,23.743,154.313
C06184=1069.627,-34.349,438.363,172.573,23.741,154.312
C06185=1069.621,-34.599,438.375,172.572,23.738,154.312
C06186=1069.615,-34.849,438.388,172.570,23.736,154.312
C06187=1069.609,-35.098,438.401,172.568,23.734,154.312
C06188=1069.603,-35.348,438.414,172.567,23.732,154.312
C06189=1069.597,-35.597,438.427,172.566,23.729,154.311
C06190=1069.590,-35.847,438.439,172.564,23.727,154.311
C06191=1069.584,-36.096,438.451,172.563,23.725,154.311
C06192=1069.578,-36.346,438.465,172.561,23.723,154.311
C06193=1069.572,-36.596,438.477,172.560,23.721,154.310
C06194=1069.567,-36.845,438.489,172.559,23.718,154.310
C06195=1069.561,-37.094,438.503,172.557,23.716,154.310
C06196=1069.555,-37.344,438.515,172.556,23.714,154.310
C06197=1069.549,-37.594,438.528,172.554,23.712,154.310
C06198=1069.543,-37.844,438.540,172.553,23.710,154.309
C06199=1069.537,-38.093,438.554,172.552,23.708,154.309
C06200=1069.531,-38.343,438.566,172.550,23.706,154.309
C06201=1069.525,-38.593,438.579,172.548,23.703,154.309
C06202=1069.519,-38.843,438.591,172.546,23.701,154.309
C06203=1069.514,-39.091,438.604,172.545,23.699,154.308
C06204=1069.507,-39.341,438.616,172.544,23.697,154.308
C06205=1069.501,-39.591,438.629,172.542,23.694,154.308
C06206=1069.495,-39.840,438.641,172.541,23.692,154.308
C06207=1069.489,-40.090,438.654,172.540,23.690,154.307
C06208=1069.482,-40.339,438.666,172.538,23.688,154.307
C06209=1069.476,-40.589,438.679,172.537,23.686,154.307
C06210=1069.470,-40.839,438.692,172.535,23.684,154.307
C06211=1069.465,-41.089,438.704,172.534,23.682,154.307
C06212=1069.458,-41.338,438.717,172.532,23.680,154.306
C06213=1069.452,-41.587,438.729,172.531,23.678,154.306
C06214=1069.446,-41.837,438.742,172.529,23.676,154.306
C06215=1069.440,-42.087,438.754,172.527,23.673,154.306
C06216=1069.434,-42.336,438.766,172.526,23.671,154.306
C06217=1069.428,-42.586,438.779,172.524,23.669,154.306
C06218=1069.422,-42.836,438.791,172.523,23.667,154.305
C06219=1069.416,-43.085,438.804,172.522,23.665,154.305
C06220=1069.410,-43.334,438.816,172.520,23.663,154.305
C06221=1069.404,-43.584,438.829,172.519,23.661,154.305
C06222=1069.398,-43.834,438.841,172.517,23.658,154.305
C06223=1069.391,-44.084,438.853,172.516,23.657,154.304
C06224=1069.385,-44.334,438.866,172.514,23.655,154.304
C06225=1069.379,-44.583,438.878,172.513,23.652,154.304
C06226=1069.374,-44.833,438.890,172.512,23.650,154.304
C06227=1069.367,-45.082,438.902,172.510,23.648,154.304
C06228=1069.362,-45.332,438.915,172.509,23.646,154.303
C06229=1069.356,-45.582,438.927,172.507,23.644,154.303
C06230=1069.349,-45.832,438.939,172.505,23.642,154.303
C06231=1069.343,-46.080,438.952,172.504,23.640,154.303
C06232=1069.337,-46.330,438.965,172.502,23.638,154.303
C06233=1069.332,-46.580,438.977,172.501,23.635,154.302
C06234=1069.325,-46.829,438.989,172.499,23.634,154.302
C06235=1069.319,-47.079,439.002,172.498,23.632,154.302
C06236=1069.314,-47.328,439.014,172.496,23.629,154.302
C06237=1069.307,-47.578,439.026,172.495,23.627,154.302
C06238=1069.301,-47.828,439.039,172.494,23.625,154.301
C06239=1069.295,-48.078,439.051,172.492,23.623,154.301
C06240=1069.289,-48.327,439.063,172.491,23.621,154.301
C06241=1069.284,-48.577,439.075,172.489,23.619,154.301
C06242=1069.278,-48.827,439.087,172.488,23.617,154.301
C06243=1069.271,-49.077,439.099,172.486,23.615,154.301
C06244=1069.266,-49.326,439.111,172.485,23.613,154.300
C06245=1069.259,-49.604,439.125,172.483,23.610,154.300
C06246=1069.252,-49.880,439.139,172.481,23.608,154.300
C06247=1069.245,-50.157,439.152,172.480,23.606,154.300
C06248=1069.238,-50.434,439.166,172.478,23.603,154.300
C06249=1069.233,-50.684,439.178,172.476,23.602,154.299
C06250=1069.226,-50.933,439.190,172.475,23.600,154.299
C06251=1069.221,-51.183,439.202,172.473,23.598,154.299
C06252=1069.214,-51.433,439.214,172.472,23.596,154.299
C06253=1069.208,-51.682,439.226,172.470,23.594,154.299
C06254=1069.202,-51.932,439.238,172.469,23.592,154.299
C06255=1069.196,-52.181,439.250,172.467,23.590,154.298
C06256=1069.190,-52.431,439.262,172.466,23.588,154.298
C06257=1069.183,-52.681,439.274,172.464,23.586,154.298
C06258=1069.177,-52.931,439.285,172.463,23.584,154.298
C06259=1069.171,-53.181,439.298,172.462,23.582,154.298
C06260=1069.165,-53.429,439.310,172.460,23.580,154.298
C06261=1069.158,-53.679,439.322,172.459,23.579,154.298
C06262=1069.152,-53.929,439.334,172.456,23.576,154.297
C06263=1069.146,-54.179,439.345,172.455,23.574,154.297
C06264=1069.140,-54.428,439.357,172.453,23.573,154.297
C06265=1069.134,-54.678,439.370,172.452,23.570,154.297
C06266=1069.127,-54.927,439.381,172.450,23.568,154.297
C06267=1069.121,-55.177,439.394,172.449,23.566,154.297
C06268=1069.116,-55.427,439.405,172.447,23.565,154.296
C06269=1069.109,-55.676,439.417,172.446,23.563,154.296
C06270=1069.103,-55.926,439.429,172.445,23.561,154.296
C06271=1069.097,-56.175,439.441,172.443,23.559,154.296
C06272=1069.091,-56.425,439.452,172.442,23.557,154.296
C06273=1069.085,-56.675,439.465,172.440,23.555,154.296
C06274=1069.078,-56.925,439.477,172.439,23.553,154.296
C06275=1069.072,-57.174,439.488,172.437,23.552,154.295
C06276=1069.066,-57.424,439.500,172.436,23.550,154.295
C06277=1069.060,-57.674,439.512,172.434,23.548,154.295
C06278=1069.054,-57.923,439.523,172.432,23.546,154.295
C06279=1069.048,-58.173,439.536,172.430,23.544,154.295
C06280=1069.042,-58.423,439.548,172.429,23.542,154.295
C06281=1069.036,-58.672,439.558,172.427,23.540,154.295
C06282=1069.029,-58.922,439.570,172.426,23.538,154.294
C06283=1069.023,-59.172,439.583,172.424,23.536,154.294
C06284=1069.017,-59.421,439.594,172.423,23.534,154.294
C06285=1069.011,-59.671,439.606,172.421,23.533,154.294
C06286=1069.005,-59.921,439.618,172.420,23.531,154.294
C06287=1068.999,-60.170,439.629,172.418,23.529,154.294
C06288=1068.993,-60.420,439.641,172.417,23.527,154.294
C06289=1068.988,-60.669,439.653,172.416,23.525,154.293
C06290=1068.981,-60.919,439.665,172.414,23.523,154.293
C06291=1068.974,-61.169,439.677,172.413,23.521,154.293
C06292=1068.969,-61.418,439.687,172.411,23.519,154.293
C06293=1068.963,-61.668,439.700,172.410,23.518,154.293
C06294=1068.956,-61.918,439.711,172.408,23.516,154.293
C06295=1068.950,-62.167,439.723,172.406,23.514,154.293
C06296=1068.944,-62.417,439.734,172.404,23.512,154.292
C06297=1068.939,-62.666,439.746,172.403,23.510,154.292
C06298=1068.932,-62.916,439.758,172.401,23.508,154.292
C06299=1068.926,-63.165,439.769,172.400,23.506,154.292
C06300=1068.920,-63.415,439.782,172.398,23.504,154.292
C06301=1068.914,-63.666,439.793,172.397,23.502,154.292
C06302=1068.908,-63.914,439.804,172.395,23.500,154.292
C06303=1068.902,-64.165,439.816,172.394,23.499,154.291
C06304=1068.896,-64.414,439.828,172.392,23.497,154.291
C06305=1068.890,-64.664,439.839,172.391,23.495,154.291
C06306=1068.884,-64.913,439.851,172.389,23.493,154.291
C06307=1068.878,-65.163,439.862,172.388,23.491,154.291
C06308=1068.873,-65.413,439.873,172.386,23.490,154.291
C06309=1068.865,-65.691,439.886,172.384,23.487,154.291
C06310=1068.859,-65.969,439.900,172.383,23.485,154.290
C06311=1068.852,-66.248,439.912,172.381,23.483,154.290
C06312=1068.845,-66.526,439.925,172.380,23.481,154.290
C06313=1068.839,-66.776,439.936,172.378,23.480,154.290
C06314=1068.833,-67.025,439.948,172.376,23.477,154.290
C06315=1068.827,-67.275,439.959,172.374,23.475,154.290
C06316=1068.821,-67.525,439.971,172.373,23.474,154.290
C06317=1068.815,-67.774,439.982,172.371,23.472,154.290
C06318=1068.809,-68.024,439.994,172.370,23.470,154.289
C06319=1068.803,-68.273,440.005,172.368,23.468,154.289
C06320=1068.796,-68.523,440.017,172.367,23.467,154.289
C06321=1068.791,-68.773,440.028,172.365,23.465,154.289
C06322=1068.785,-69.023,440.040,172.364,23.463,154.289
C06323=1068.779,-69.272,440.051,172.362,23.461,154.289
C06324=1068.773,-69.522,440.062,172.361,23.460,154.289
C06325=1068.767,-69.771,440.074,172.359,23.458,154.289
C06326=1068.761,-70.022,440.086,172.358,23.456,154.288
C06327=1068.755,-70.271,440.096,172.356,23.454,154.288
C06328=1068.749,-70.521,440.108,172.355,23.452,154.288
C06329=1068.743,-70.770,440.119,172.353,23.450,154.288
C06330=1068.737,-71.020,440.130,172.352,23.449,154.288
C06331=1068.731,-71.270,440.143,172.350,23.447,154.288
C06332=1068.726,-71.519,440.154,172.349,23.445,154.288
C06333=1068.719,-71.769,440.165,172.347,23.443,154.288
C06334=1068.713,-72.019,440.176,172.345,23.441,154.287
C06335=1068.707,-72.268,440.188,172.343,23.440,154.287
C06336=1068.701,-72.518,440.199,172.342,23.438,154.287
C06337=1068.696,-72.768,440.210,172.340,23.436,154.287
C06338=1068.690,-73.018,440.221,172.339,23.434,154.287
C06339=1068.684,-73.267,440.233,172.337,23.432,154.287
C06340=1068.677,-73.517,440.244,172.336,23.431,154.287
C06341=1068.672,-73.766,440.255,172.334,23.429,154.287
C06342=1068.666,-74.016,440.266,172.333,23.427,154.287
C06343=1068.660,-74.266,440.277,172.331,23.425,154.286
C06344=1068.653,-74.515,440.289,172.330,23.424,154.286
C06345=1068.647,-74.765,440.300,172.328,23.422,154.286
C06346=1068.641,-75.015,440.311,172.327,23.421,154.286
C06347=1068.635,-75.265,440.322,172.325,23.419,154.286
C06348=1068.629,-75.514,440.333,172.324,23.417,154.286
C06349=1068.624,-75.764,440.344,172.322,23.416,154.286
C06350=1068.617,-76.013,440.356,172.321,23.414,154.286
C06351=1068.611,-76.263,440.367,172.319,23.413,154.286
C06352=1068.605,-76.513,440.378,172.317,23.411,154.286
C06353=1068.599,-76.763,440.389,172.316,23.409,154.285
C06354=1068.593,-77.012,440.399,172.314,23.408,154.285
C06355=1068.586,-77.262,440.410,172.313,23.406,154.285
C06356=1068.581,-77.511,440.421,172.311,23.405,154.285
C06357=1068.574,-77.762,440.432,172.309,23.402,154.285
C06358=1068.568,-78.011,440.443,172.307,23.400,154.285
C06359=1068.562,-78.260,440.455,172.306,23.399,154.285
C06360=1068.556,-78.510,440.466,172.304,23.397,154.285
C06361=1068.550,-78.760,440.477,172.303,23.396,154.285
C06362=1068.544,-79.010,440.488,172.301,23.394,154.285
C06363=1068.538,-79.259,440.499,172.299,23.393,154.285
C06364=1068.533,-79.509,440.510,172.298,23.391,154.285
C06365=1068.525,-79.759,440.521,172.296,23.390,154.285
C06366=1068.520,-80.008,440.532,172.295,23.388,154.284
C06367=1068.514,-80.258,440.542,172.293,23.386,154.284
C06368=1068.508,-80.508,440.554,172.292,23.384,154.284
C06369=1068.501,-80.757,440.564,172.290,23.383,154.284
C06370=1068.495,-81.007,440.575,172.289,23.381,154.284
C06371=1068.489,-81.257,440.586,172.287,23.380,154.284
C06372=1068.483,-81.506,440.597,172.285,23.379,154.284
C06373=1068.475,-81.787,440.609,172.284,23.377,154.284
C06374=1068.469,-82.067,440.621,172.281,23.375,154.284
C06375=1068.463,-82.348,440.633,172.280,23.373,154.284
C06376=1068.455,-82.629,440.645,172.278,23.371,154.284
C06377=1068.449,-82.878,440.656,172.277,23.370,154.284
C06378=1068.443,-83.128,440.667,172.275,23.369,154.284
C06379=1068.436,-83.378,440.678,172.274,23.367,154.283
C06380=1068.430,-83.627,440.689,172.272,23.366,154.283
C06381=1068.425,-83.877,440.699,172.270,23.364,154.283
C06382=1068.417,-84.127,440.710,172.269,23.362,154.283
C06383=1068.412,-84.376,440.721,172.267,23.361,154.283
C06384=1068.406,-84.626,440.731,172.266,23.360,154.283
C06385=1068.399,-84.876,440.742,172.264,23.358,154.283
C06386=1068.394,-85.126,440.753,172.262,23.356,154.283
C06387=1068.388,-85.375,440.764,172.260,23.355,154.283
C06388=1068.381,-85.625,440.774,172.259,23.353,154.283
C06389=1068.375,-85.874,440.785,172.257,23.352,154.283
C06390=1068.369,-86.124,440.796,172.255,23.350,154.283
C06391=1068.362,-86.374,440.807,172.254,23.349,154.283
C06392=1068.357,-86.624,440.817,172.252,23.347,154.283
C06393=1068.351,-86.873,440.828,172.251,23.346,154.283
C06394=1068.344,-87.123,440.838,172.249,23.345,154.283
C06395=1068.338,-87.373,440.849,172.247,23.343,154.283
C06396=1068.332,-87.622,440.860,172.246,23.341,154.283
C06397=1068.326,-87.872,440.870,172.244,23.340,154.283
C06398=1068.320,-88.122,440.881,172.243,23.338,154.282
C06399=1068.313,-88.371,440.891,172.241,23.337,154.282
C06400=1068.308,-88.621,440.902,172.239,23.336,154.282
C06401=1068.302,-88.870,440.913,172.238,23.334,154.282
C06402=1068.295,-89.121,440.923,172.236,23.332,154.282
C06403=1068.289,-89.370,440.934,172.235,23.331,154.282
C06404=1068.284,-89.620,440.945,172.233,23.330,154.282
C06405=1068.277,-89.869,440.955,172.231,23.328,154.282
C06406=1068.271,-90.120,440.965,172.230,23.327,154.282
C06407=1068.265,-90.369,440.976,172.228,23.325,154.282
C06408=1068.259,-90.619,440.987,172.227,23.324,154.282
C06409=1068.254,-90.869,440.997,172.225,23.323,154.282
C06410=1068.247,-91.118,441.007,172.223,23.321,154.282
C06411=1068.241,-91.368,441.018,172.222,23.319,154.282
C06412=1068.234,-91.617,441.029,172.220,23.318,154.282
C06413=1068.229,-91.867,441.039,172.219,23.317,154.282
C06414=1068.223,-92.117,441.050,172.217,23.316,154.282
C06415=1068.217,-92.366,441.060,172.215,23.314,154.282
C06416=1068.211,-92.617,441.070,172.214,23.313,154.282
C06417=1068.204,-92.866,441.081,172.212,23.311,154.282
C06418=1068.198,-93.116,441.092,172.211,23.310,154.282
C06419=1068.193,-93.366,441.102,172.209,23.308,154.282
C06420=1068.186,-93.615,441.112,172.207,23.307,154.282
C06421=1068.180,-93.866,441.122,172.206,23.306,154.282
C06422=1068.174,-94.115,441.133,172.204,23.304,154.282
C06423=1068.168,-94.364,441.144,172.203,23.303,154.281
C06424=1068.162,-94.614,441.153,172.201,23.301,154.281
C06425=1068.156,-94.864,441.164,172.199,23.300,154.281
C06426=1068.151,-95.114,441.174,172.198,23.299,154.281
C06427=1068.144,-95.363,441.185,172.196,23.297,154.281
C06428=1068.138,-95.613,441.196,172.194,23.296,154.281
C06429=1068.132,-95.863,441.205,172.193,23.295,154.281
C06430=1068.126,-96.112,441.216,172.191,23.293,154.281
C06431=1068.120,-96.362,441.226,172.189,23.292,154.281
C06432=1068.114,-96.612,441.237,172.188,23.290,154.281
C06433=1068.108,-96.861,441.246,172.186,23.289,154.281
C06434=1068.102,-97.111,441.257,172.185,23.288,154.281
C06435=1068.096,-97.361,441.267,172.183,23.286,154.281
C06436=1068.090,-97.611,441.278,172.181,23.285,154.281
C06437=1068.083,-97.893,441.289,172.179,23.283,154.281
C06438=1068.076,-98.176,441.301,172.177,23.282,154.281
C06439=1068.069,-98.459,441.313,172.176,23.281,154.281
C06440=1068.062,-98.741,441.324,172.173,23.279,154.281
C06441=1068.055,-98.992,441.334,172.171,23.278,154.281
C06442=1068.050,-99.241,441.345,172.170,23.276,154.281
C06443=1068.044,-99.491,441.354,172.168,23.275,154.281
C06444=1068.037,-99.740,441.365,172.167,23.274,154.281
C06445=1068.032,-99.991,441.375,172.165,23.272,154.281
C06446=1068.025,-100.240,441.385,172.163,23.272,154.281
C06447=1068.019,-100.489,441.395,172.161,23.270,154.281
C06448=1068.014,-100.740,441.405,172.160,23.269,154.281
C06449=1068.006,-100.989,441.415,172.158,23.268,154.281
C06450=1068.000,-101.239,441.425,172.157,23.266,154.281
C06451=1067.995,-101.489,441.436,172.155,23.265,154.281
C06452=1067.988,-101.739,441.445,172.153,23.264,154.281
C06453=1067.982,-101.988,441.455,172.152,23.262,154.281
C06454=1067.977,-102.238,441.466,172.150,23.262,154.281
C06455=1067.970,-102.488,441.475,172.148,23.260,154.281
C06456=1067.964,-102.737,441.486,172.147,23.259,154.281
C06457=1067.958,-102.987,441.495,172.145,23.258,154.281
C06458=1067.952,-103.237,441.505,172.143,23.256,154.281
C06459=1067.946,-103.486,441.516,172.142,23.255,154.281
C06460=1067.939,-103.736,441.526,172.140,23.254,154.281
C06461=1067.934,-103.987,441.536,172.138,23.253,154.281
C06462=1067.927,-104.236,441.546,172.137,23.252,154.281
C06463=1067.921,-104.486,441.556,172.135,23.250,154.281
C06464=1067.915,-104.735,441.565,172.133,23.249,154.281
C06465=1067.909,-104.985,441.576,172.131,23.248,154.281
C06466=1067.903,-105.235,441.586,172.130,23.247,154.281
C06467=1067.897,-105.484,441.595,172.129,23.246,154.281
C06468=1067.890,-105.734,441.605,172.127,23.245,154.281
C06469=1067.885,-105.984,441.616,172.126,23.244,154.281
C06470=1067.879,-106.233,441.625,172.124,23.243,154.281
C06471=1067.872,-106.483,441.635,172.122,23.241,154.281
C06472=1067.866,-106.732,441.645,172.121,23.240,154.281
C06473=1067.860,-106.983,441.655,172.119,23.239,154.281
C06474=1067.854,-107.232,441.665,172.117,23.238,154.281
C06475=1067.848,-107.482,441.674,172.116,23.237,154.281
C06476=1067.842,-107.732,441.684,172.114,23.235,154.281
C06477=1067.835,-107.981,441.694,172.112,23.235,154.281
C06478=1067.829,-108.231,441.704,172.111,23.233,154.281
C06479=1067.824,-108.481,441.714,172.109,23.233,154.282
C06480=1067.818,-108.731,441.724,172.107,23.231,154.282
C06481=1067.811,-108.980,441.734,172.106,23.230,154.282
C06482=1067.805,-109.230,441.743,172.104,23.229,154.282
C06483=1067.799,-109.480,441.753,172.102,23.228,154.282
C06484=1067.793,-109.729,441.763,172.100,23.227,154.282
C06485=1067.787,-109.979,441.772,172.099,23.226,154.282
C06486=1067.780,-110.229,441.782,172.097,23.225,154.282
C06487=1067.774,-110.478,441.792,172.095,23.224,154.282
C06488=1067.768,-110.728,441.802,172.094,23.222,154.282
C06489=1067.762,-110.978,441.812,172.092,23.221,154.282
C06490=1067.756,-111.228,441.821,172.090,23.220,154.282
C06491=1067.750,-111.478,441.831,172.088,23.219,154.282
C06492=1067.744,-111.727,441.840,172.087,23.218,154.282
C06493=1067.738,-111.977,441.850,172.085,23.217,154.282
C06494=1067.731,-112.227,441.860,172.083,23.216,154.282
C06495=1067.725,-112.476,441.870,172.082,23.215,154.282
C06496=1067.719,-112.726,441.879,172.080,23.214,154.282
C06497=1067.713,-112.976,441.889,172.078,23.213,154.282
C06498=1067.706,-113.226,441.899,172.076,23.212,154.282
C06499=1067.700,-113.475,441.908,172.075,23.211,154.282
C06500=1067.695,-113.726,441.918,172.073,23.210,154.282
C06501=1067.688,-114.006,441.929,172.071,23.209,154.282
C06502=1067.681,-114.287,441.940,172.070,23.207,154.282
C06503=1067.674,-114.567,441.950,172.067,23.206,154.283
C06504=1067.667,-114.848,441.961,172.065,23.205,154.283
C06505=1067.661,-115.097,441.970,172.063,23.204,154.283
C06506=1067.655,-115.347,441.980,172.062,23.203,154.283
C06507=1067.648,-115.597,441.990,172.060,23.202,154.283
C06508=1067.642,-115.847,441.999,172.058,23.201,154.283
C06509=1067.636,-116.097,442.009,172.057,23.200,154.283
C06510=1067.630,-116.346,442.018,172.055,23.199,154.283
C06511=1067.624,-116.596,442.028,172.053,23.198,154.283
C06512=1067.618,-116.846,442.037,172.052,23.198,154.283
C06513=1067.611,-117.096,442.047,172.050,23.197,154.283
C06514=1067.605,-117.346,442.057,172.049,23.196,154.283
C06515=1067.599,-117.595,442.066,172.047,23.195,154.283
C06516=1067.594,-117.845,442.075,172.045,23.194,154.283
C06517=1067.588,-118.095,442.084,172.044,23.193,154.283
C06518=1067.581,-118.345,442.094,172.042,23.192,154.283
C06519=1067.575,-118.595,442.103,172.040,23.191,154.283
C06520=1067.569,-118.844,442.113,172.038,23.190,154.284
C06521=1067.562,-119.094,442.122,172.036,23.189,154.284
C06522=1067.556,-119.344,442.131,172.035,23.188,154.284
C06523=1067.550,-119.593,442.141,172.033,23.187,154.284
C06524=1067.544,-119.843,442.151,172.031,23.187,154.284
C06525=1067.538,-120.092,442.160,172.029,23.186,154.284
C06526=1067.532,-120.342,442.169,172.028,23.184,154.284
C06527=1067.526,-120.593,442.178,172.026,23.184,154.284
C06528=1067.520,-120.842,442.188,172.024,23.183,154.284
C06529=1067.514,-121.092,442.197,172.023,23.182,154.284
C06530=1067.507,-121.342,442.206,172.021,23.181,154.284
C06531=1067.501,-121.591,442.216,172.019,23.180,154.284
C06532=1067.495,-121.840,442.225,172.017,23.179,154.285
C06533=1067.489,-122.091,442.234,172.016,23.178,154.284
C06534=1067.483,-122.341,442.243,172.014,23.177,154.285
C06535=1067.477,-122.591,442.253,172.012,23.177,154.285
C06536=1067.471,-122.840,442.263,172.011,23.176,154.285
C06537=1067.464,-123.090,442.272,172.009,23.175,154.285
C06538=1067.458,-123.339,442.281,172.008,23.174,154.285
C06539=1067.452,-123.589,442.290,172.006,23.173,154.285
C06540=1067.446,-123.839,442.299,172.004,23.173,154.285
C06541=1067.440,-124.089,442.309,172.002,23.172,154.285
C06542=1067.434,-124.339,442.318,172.000,23.171,154.285
C06543=1067.427,-124.589,442.327,171.999,23.170,154.285
C06544=1067.422,-124.838,442.336,171.997,23.169,154.285
C06545=1067.415,-125.088,442.345,171.995,23.168,154.286
C06546=1067.409,-125.338,442.355,171.993,23.168,154.286
C06547=1067.403,-125.588,442.363,171.991,23.167,154.286
C06548=1067.397,-125.837,442.373,171.990,23.166,154.286
C06549=1067.391,-126.087,442.382,171.988,23.165,154.286
C06550=1067.384,-126.337,442.390,171.986,23.165,154.286
C06551=1067.378,-126.586,442.400,171.984,23.164,154.286
C06552=1067.372,-126.836,442.409,171.982,23.163,154.286
C06553=1067.366,-127.086,442.419,171.981,23.162,154.286
C06554=1067.360,-127.335,442.427,171.980,23.162,154.287
C06555=1067.354,-127.585,442.436,171.978,23.161,154.287
C06556=1067.347,-127.835,442.446,171.976,23.160,154.287
C06557=1067.342,-128.086,442.455,171.974,23.159,154.287
C06558=1067.339,-128.336,442.466,171.973,23.157,154.287
C06559=1067.337,-128.587,442.476,171.972,23.155,154.286
C06560=1067.338,-128.838,442.488,171.971,23.151,154.286
C06561=1067.340,-129.091,442.502,171.970,23.148,154.285
C06562=1067.343,-129.343,442.515,171.969,23.143,154.285
C06563=1067.349,-129.595,442.529,171.969,23.138,154.284
C06564=1067.357,-129.844,442.545,171.969,23.132,154.283
C06565=1066.969,-129.867,442.370,171.922,23.279,154.315
C06566=1066.961,-129.616,442.355,171.921,23.284,154.316
C06567=1066.956,-129.365,442.341,171.922,23.289,154.317
C06568=1066.953,-129.114,442.327,171.923,23.294,154.318
C06569=1066.951,-128.860,442.314,171.923,23.298,154.319
C06570=1066.950,-128.610,442.302,171.925,23.301,154.319
C06571=1066.952,-128.360,442.291,171.926,23.304,154.319
C06572=1066.955,-128.108,442.281,171.927,23.306,154.320
C06573=1066.960,-127.857,442.271,171.929,23.306,154.319
C06574=1066.966,-127.608,442.262,171.931,23.308,154.319
C06575=1066.972,-127.359,442.252,171.932,23.308,154.319
C06576=1066.978,-127.108,442.244,171.933,23.309,154.319
C06577=1066.984,-126.858,442.234,171.935,23.310,154.319
C06578=1066.991,-126.609,442.225,171.937,23.310,154.319
C06579=1066.997,-126.359,442.216,171.939,23.311,154.319
C06580=1067.002,-126.109,442.207,171.941,23.312,154.319
C06581=1067.009,-125.860,442.198,171.942,23.312,154.319
C06582=1067.016,-125.610,442.188,171.944,23.313,154.319
C06583=1067.021,-125.360,442.180,171.946,23.314,154.318
C06584=1067.028,-125.110,442.170,171.948,23.315,154.318
C06585=1067.034,-124.861,442.161,171.950,23.315,154.318
C06586=1067.040,-124.611,442.152,171.951,23.317,154.318
C06587=1067.046,-124.361,442.143,171.953,23.318,154.318
C06588=1067.052,-124.111,442.133,171.955,23.318,154.318
C06589=1067.059,-123.862,442.124,171.957,23.319,154.318
C06590=1067.065,-123.612,442.115,171.959,23.320,154.318
C06591=1067.070,-123.362,442.106,171.960,23.320,154.318
C06592=1067.077,-123.112,442.097,171.962,23.322,154.318
C06593=1067.083,-122.863,442.087,171.964,23.323,154.318
C06594=1067.089,-122.613,442.078,171.966,23.323,154.317
C06595=1067.095,-122.363,442.068,171.967,23.324,154.317
C06596=1067.101,-122.114,442.060,171.968,23.325,154.317
C06597=1067.107,-121.864,442.051,171.970,23.326,154.317
C06598=1067.113,-121.614,442.041,171.972,23.326,154.317
C06599=1067.120,-121.364,442.032,171.974,23.327,154.317
C06600=1067.126,-121.114,442.022,171.975,23.328,154.317
C06601=1067.132,-120.865,442.012,171.977,23.329,154.317
C06602=1067.138,-120.614,442.004,171.979,23.330,154.317
C06603=1067.144,-120.365,441.995,171.981,23.331,154.317
C06604=1067.150,-120.116,441.985,171.982,23.332,154.317
C06605=1067.156,-119.866,441.976,171.984,23.333,154.317
C06606=1067.163,-119.616,441.966,171.986,23.333,154.317
C06607=1067.169,-119.366,441.957,171.988,23.335,154.317
C06608=1067.175,-119.116,441.947,171.989,23.336,154.316
C06609=1067.181,-118.867,441.938,171.991,23.336,154.316
C06610=1067.187,-118.617,441.928,171.993,23.338,154.316
C06611=1067.193,-118.367,441.918,171.995,23.338,154.316
C06612=1067.199,-118.117,441.910,171.996,23.339,154.316
C06613=1067.206,-117.868,441.901,171.998,23.340,154.316
C06614=1067.212,-117.618,441.891,172.000,23.341,154.316
C06615=1067.218,-117.368,441.882,172.002,23.342,154.316
C06616=1067.224,-117.118,441.872,172.003,23.343,154.316
C06617=1067.230,-116.869,441.863,172.005,23.344,154.316
C06618=1067.237,-116.619,441.853,172.007,23.345,154.316
C06619=1067.243,-116.369,441.844,172.009,23.346,154.316
C06620=1067.249,-116.119,441.834,172.010,23.347,154.316
C06621=1067.255,-115.869,441.824,172.012,23.348,154.316
C06622=1067.261,-115.620,441.815,172.014,23.349,154.315
C06623=1067.267,-115.371,441.806,172.015,23.350,154.316
C06624=1067.273,-115.121,441.796,172.017,23.351,154.315
C06625=1067.279,-114.871,441.787,172.018,23.352,154.315
C06626=1067.286,-114.590,441.775,172.021,23.353,154.315
C06627=1067.293,-114.309,441.765,172.022,23.354,154.315
C06628=1067.300,-114.028,441.754,172.024,23.355,154.315
C06629=1067.307,-113.748,441.743,172.026,23.356,154.315
C06630=1067.313,-113.498,441.733,172.028,23.357,154.315
C06631=1067.319,-113.248,441.724,172.029,23.358,154.315
C06632=1067.325,-112.998,441.714,172.031,23.359,154.315
C06633=1067.332,-112.749,441.705,172.033,23.360,154.315
C06634=1067.338,-112.499,441.695,172.035,23.361,154.315
C06635=1067.344,-112.249,441.686,172.036,23.362,154.315
C06636=1067.349,-111.999,441.675,172.038,23.364,154.315
C06637=1067.356,-111.749,441.666,172.040,23.364,154.315
C06638=1067.362,-111.499,441.656,172.041,23.366,154.315
C06639=1067.368,-111.250,441.646,172.043,23.366,154.315
C06640=1067.374,-111.000,441.636,172.045,23.368,154.315
C06641=1067.381,-110.751,441.627,172.047,23.368,154.315
C06642=1067.387,-110.501,441.617,172.048,23.370,154.315
C06643=1067.393,-110.251,441.608,172.050,23.371,154.315
C06644=1067.399,-110.001,441.598,172.052,23.372,154.315
C06645=1067.406,-109.752,441.588,172.053,23.373,154.315
C06646=1067.411,-109.502,441.578,172.055,23.374,154.314
C06647=1067.417,-109.252,441.568,172.057,23.375,154.314
C06648=1067.423,-109.002,441.559,172.058,23.376,154.314
C06649=1067.429,-108.752,441.549,172.060,23.377,154.314
C06650=1067.436,-108.503,441.539,172.062,23.378,154.314
C06651=1067.442,-108.254,441.529,172.063,23.380,154.314
C06652=1067.448,-108.004,441.520,172.065,23.381,154.314
C06653=1067.454,-107.754,441.510,172.067,23.382,154.314
C06654=1067.461,-107.504,441.500,172.069,23.383,154.314
C06655=1067.466,-107.255,441.490,172.070,23.384,154.314
C06656=1067.473,-107.005,441.480,172.072,23.385,154.314
C06657=1067.479,-106.755,441.470,172.074,23.387,154.314
C06658=1067.485,-106.505,441.461,172.075,23.387,154.314
C06659=1067.491,-106.256,441.450,172.077,23.389,154.314
C06660=1067.497,-106.006,441.440,172.079,23.390,154.314
C06661=1067.503,-105.756,441.431,172.080,23.391,154.314
C06662=1067.509,-105.506,441.421,172.082,23.392,154.314
C06663=1067.515,-105.257,441.410,172.084,23.393,154.314
C06664=1067.521,-105.007,441.401,172.086,23.395,154.314
C06665=1067.527,-104.757,441.391,172.087,23.396,154.314
C06666=1067.534,-104.507,441.381,172.089,23.397,154.314
C06667=1067.540,-104.257,441.370,172.091,23.398,154.314
C06668=1067.546,-104.007,441.361,172.092,23.399,154.314
C06669=1067.552,-103.758,441.351,172.094,23.400,154.314
C06670=1067.559,-103.508,441.341,172.096,23.402,154.314
C06671=1067.564,-103.258,441.331,172.097,23.403,154.314
C06672=1067.570,-103.009,441.321,172.099,23.404,154.314
C06673=1067.577,-102.759,441.311,172.101,23.405,154.314
C06674=1067.582,-102.509,441.301,172.102,23.406,154.314
C06675=1067.589,-102.260,441.291,172.104,23.408,154.314
C06676=1067.595,-102.010,441.281,172.106,23.409,154.314
C06677=1067.600,-101.761,441.270,172.107,23.410,154.314
C06678=1067.607,-101.511,441.261,172.109,23.412,154.314
C06679=1067.613,-101.261,441.251,172.110,23.413,154.314
C06680=1067.619,-101.011,441.240,172.112,23.414,154.314
C06681=1067.625,-100.761,441.230,172.114,23.415,154.314
C06682=1067.632,-100.512,441.220,172.116,23.416,154.314
C06683=1067.637,-100.262,441.210,172.117,23.418,154.314
C06684=1067.644,-100.013,441.199,172.119,23.419,154.314
C06685=1067.650,-99.763,441.190,172.121,23.420,154.314
C06686=1067.655,-99.513,441.180,172.122,23.422,154.314
C06687=1067.662,-99.263,441.169,172.124,23.423,154.314
C06688=1067.669,-99.013,441.160,172.125,23.424,154.314
C06689=1067.674,-98.764,441.149,172.127,23.425,154.314
C06690=1067.681,-98.481,441.137,172.129,23.427,154.314
C06691=1067.688,-98.198,441.126,172.130,23.428,154.314
C06692=1067.695,-97.915,441.114,172.133,23.430,154.314
C06693=1067.702,-97.632,441.103,172.135,23.431,154.314
C06694=1067.709,-97.383,441.093,172.136,23.432,154.314
C06695=1067.714,-97.133,441.083,172.138,23.434,154.314
C06696=1067.720,-96.883,441.072,172.139,23.435,154.314
C06697=1067.726,-96.634,441.061,172.141,23.436,154.314
C06698=1067.733,-96.383,441.051,172.143,23.438,154.314
C06699=1067.739,-96.134,441.041,172.144,23.439,154.314
C06700=1067.744,-95.884,441.030,172.146,23.440,154.314
C06701=1067.751,-95.635,441.020,172.148,23.442,154.314
C06702=1067.756,-95.385,441.010,172.149,23.443,154.314
C06703=1067.763,-95.135,441.000,172.151,23.445,154.314
C06704=1067.768,-94.886,440.989,172.152,23.446,154.314
C06705=1067.775,-94.635,440.979,172.154,23.447,154.314
C06706=1067.781,-94.386,440.968,172.156,23.449,154.314
C06707=1067.787,-94.136,440.958,172.157,23.450,154.314
C06708=1067.793,-93.887,440.948,172.159,23.452,154.315
C06709=1067.798,-93.637,440.937,172.161,23.453,154.315
C06710=1067.805,-93.387,440.927,172.162,23.454,154.315
C06711=1067.811,-93.137,440.916,172.164,23.456,154.315
C06712=1067.817,-92.888,440.906,172.165,23.457,154.315
C06713=1067.823,-92.638,440.895,172.167,23.458,154.315
C06714=1067.829,-92.389,440.885,172.169,23.460,154.315
C06715=1067.835,-92.139,440.874,172.170,23.461,154.315
C06716=1067.841,-91.888,440.864,172.172,23.463,154.315
C06717=1067.848,-91.639,440.853,172.174,23.464,154.315
C06718=1067.853,-91.390,440.843,172.175,23.465,154.315
C06719=1067.860,-91.140,440.833,172.177,23.467,154.315
C06720=1067.865,-90.890,440.822,172.178,23.469,154.315
C06721=1067.872,-90.640,440.811,172.180,23.470,154.315
C06722=1067.878,-90.391,440.801,172.182,23.471,154.315
C06723=1067.884,-90.141,440.790,172.184,23.473,154.315
C06724=1067.889,-89.891,440.780,172.186,23.475,154.315
C06725=1067.896,-89.642,440.769,172.187,23.476,154.315
C06726=1067.902,-89.391,440.759,172.189,23.477,154.315
C06727=1067.908,-89.142,440.748,172.191,23.479,154.315
C06728=1067.914,-88.893,440.738,172.192,23.481,154.315
C06729=1067.920,-88.643,440.726,172.194,23.482,154.315
C06730=1067.927,-88.393,440.716,172.195,23.483,154.315
C06731=1067.932,-88.143,440.706,172.197,23.484,154.315
C06732=1067.938,-87.894,440.695,172.198,23.486,154.316
C06733=1067.945,-87.644,440.684,172.200,23.488,154.316
C06734=1067.951,-87.394,440.674,172.202,23.489,154.316
C06735=1067.957,-87.145,440.663,172.203,23.491,154.316
C06736=1067.963,-86.895,440.653,172.205,23.492,154.316
C06737=1067.969,-86.645,440.642,172.206,23.493,154.316
C06738=1067.976,-86.396,440.632,172.208,23.495,154.316
C06739=1067.981,-86.146,440.621,172.210,23.497,154.316
C06740=1067.988,-85.896,440.609,172.211,23.498,154.316
C06741=1067.994,-85.647,440.599,172.213,23.499,154.316
C06742=1068.000,-85.397,440.589,172.214,23.501,154.316
C06743=1068.006,-85.147,440.578,172.216,23.502,154.316
C06744=1068.012,-84.897,440.567,172.218,23.504,154.316
C06745=1068.018,-84.648,440.557,172.219,23.506,154.316
C06746=1068.024,-84.398,440.545,172.221,23.507,154.316
C06747=1068.031,-84.149,440.535,172.222,23.508,154.316
C06748=1068.037,-83.899,440.524,172.224,23.510,154.316
C06749=1068.043,-83.649,440.513,172.226,23.511,154.316
C06750=1068.049,-83.400,440.503,172.227,23.513,154.316
C06751=1068.055,-83.150,440.492,172.229,23.514,154.317
C06752=1068.062,-82.900,440.481,172.230,23.516,154.317
C06753=1068.067,-82.651,440.470,172.232,23.518,154.317
C06754=1068.074,-82.370,440.459,172.234,23.519,154.317
C06755=1068.081,-82.089,440.446,172.236,23.521,154.317
C06756=1068.088,-81.809,440.433,172.237,23.522,154.317
C06757=1068.096,-81.528,440.421,172.240,23.525,154.317
C06758=1068.101,-81.278,440.411,172.241,23.526,154.317
C06759=1068.107,-81.028,440.400,172.243,23.528,154.317
C06760=1068.114,-80.778,440.390,172.245,23.529,154.317
C06761=1068.120,-80.529,440.379,172.246,23.530,154.317
C06762=1068.127,-80.279,440.367,172.248,23.532,154.317
C06763=1068.132,-80.030,440.356,172.249,23.534,154.317
C06764=1068.139,-79.781,440.346,172.251,23.536,154.317
C06765=1068.145,-79.530,440.334,172.253,23.537,154.317
C06766=1068.151,-79.281,440.323,172.254,23.539,154.318
C06767=1068.157,-79.031,440.312,172.256,23.540,154.318
C06768=1068.163,-78.781,440.301,172.257,23.542,154.318
C06769=1068.169,-78.532,440.290,172.259,23.544,154.318
C06770=1068.175,-78.282,440.279,172.260,23.545,154.318
C06771=1068.181,-78.032,440.268,172.262,23.547,154.318
C06772=1068.187,-77.783,440.257,172.263,23.548,154.318
C06773=1068.193,-77.532,440.246,172.265,23.550,154.318
C06774=1068.199,-77.283,440.235,172.267,23.551,154.318
C06775=1068.206,-77.033,440.225,172.268,23.553,154.318
C06776=1068.212,-76.784,440.213,172.269,23.555,154.319
C06777=1068.218,-76.535,440.202,172.271,23.556,154.319
C06778=1068.224,-76.285,440.191,172.273,23.558,154.319
C06779=1068.230,-76.035,440.180,172.274,23.560,154.319
C06780=1068.236,-75.785,440.169,172.276,23.561,154.319
C06781=1068.242,-75.535,440.158,172.277,23.563,154.319
C06782=1068.248,-75.285,440.147,172.280,23.565,154.319
C06783=1068.254,-75.036,440.135,172.281,23.567,154.319
C06784=1068.260,-74.787,440.124,172.283,23.569,154.319
C06785=1068.266,-74.537,440.113,172.284,23.570,154.319
C06786=1068.272,-74.287,440.102,172.286,23.572,154.319
C06787=1068.278,-74.037,440.091,172.287,23.574,154.320
C06788=1068.284,-73.788,440.079,172.289,23.575,154.320
C06789=1068.291,-73.538,440.068,172.290,23.577,154.320
C06790=1068.296,-73.288,440.057,172.292,23.579,154.320
C06791=1068.302,-73.039,440.046,172.293,23.581,154.320
C06792=1068.308,-72.789,440.035,172.295,23.582,154.320
C06793=1068.314,-72.540,440.023,172.297,23.584,154.320
C06794=1068.320,-72.289,440.012,172.298,23.586,154.320
C06795=1068.326,-72.040,440.001,172.300,23.588,154.320
C06796=1068.332,-71.791,439.989,172.301,23.589,154.321
C06797=1068.338,-71.541,439.978,172.302,23.591,154.321
C06798=1068.344,-71.291,439.967,172.304,23.593,154.321
C06799=1068.350,-71.041,439.955,172.306,23.594,154.321
C06800=1068.356,-70.792,439.944,172.307,23.596,154.321
C06801=1068.362,-70.542,439.932,172.309,23.598,154.321
C06802=1068.368,-70.292,439.922,172.310,23.600,154.321
C06803=1068.374,-70.043,439.910,172.312,23.602,154.322
C06804=1068.380,-69.793,439.899,172.314,23.604,154.321
C06805=1068.385,-69.543,439.887,172.316,23.605,154.322
C06806=1068.392,-69.294,439.875,172.317,23.607,154.322
C06807=1068.397,-69.044,439.864,172.319,23.609,154.322
C06808=1068.404,-68.794,439.853,172.320,23.611,154.322
C06809=1068.410,-68.545,439.842,172.322,23.613,154.322
C06810=1068.415,-68.295,439.830,172.323,23.615,154.322
C06811=1068.421,-68.045,439.819,172.325,23.616,154.322
C06812=1068.428,-67.796,439.807,172.326,23.618,154.322
C06813=1068.434,-67.546,439.796,172.328,23.620,154.323
C06814=1068.439,-67.296,439.783,172.329,23.622,154.323
C06815=1068.445,-67.047,439.773,172.331,23.623,154.323
C06816=1068.452,-66.797,439.761,172.332,23.625,154.323
C06817=1068.458,-66.548,439.750,172.334,23.627,154.323
C06818=1068.464,-66.269,439.737,172.335,23.629,154.323
C06819=1068.471,-65.991,439.724,172.337,23.631,154.323
C06820=1068.478,-65.712,439.711,172.339,23.633,154.324
C06821=1068.484,-65.433,439.698,172.340,23.635,154.324
C06822=1068.491,-65.184,439.686,172.342,23.637,154.324
C06823=1068.497,-64.934,439.675,172.343,23.639,154.324
C06824=1068.503,-64.684,439.664,172.346,23.641,154.324
C06825=1068.508,-64.435,439.652,172.347,23.643,154.324
C06826=1068.515,-64.185,439.640,172.349,23.645,154.324
C06827=1068.521,-63.936,439.629,172.350,23.647,154.325
C06828=1068.527,-63.686,439.618,172.352,23.648,154.325
C06829=1068.533,-63.436,439.605,172.353,23.650,154.325
C06830=1068.539,-63.187,439.593,172.355,23.652,154.325
C06831=1068.545,-62.937,439.582,172.356,23.654,154.325
C06832=1068.551,-62.688,439.571,172.358,23.656,154.325
C06833=1068.557,-62.437,439.559,172.359,23.658,154.325
C06834=1068.563,-62.189,439.547,172.361,23.660,154.326
C06835=1068.569,-61.938,439.536,172.362,23.661,154.326
C06836=1068.576,-61.689,439.524,172.364,23.663,154.326
C06837=1068.581,-61.439,439.513,172.365,23.665,154.326
C06838=1068.588,-61.189,439.501,172.367,23.667,154.326
C06839=1068.594,-60.940,439.489,172.368,23.669,154.326
C06840=1068.599,-60.690,439.477,172.370,23.671,154.326
C06841=1068.606,-60.440,439.465,172.371,23.673,154.327
C06842=1068.612,-60.191,439.454,172.373,23.675,154.327
C06843=1068.618,-59.941,439.442,172.375,23.677,154.327
C06844=1068.624,-59.692,439.430,172.376,23.679,154.327
C06845=1068.630,-59.442,439.419,172.378,23.680,154.327
C06846=1068.636,-59.192,439.407,172.379,23.682,154.327
C06847=1068.642,-58.943,439.394,172.381,23.684,154.327
C06848=1068.648,-58.693,439.383,172.382,23.686,154.328
C06849=1068.655,-58.444,439.372,172.384,23.688,154.328
C06850=1068.661,-58.194,439.359,172.385,23.690,154.328
C06851=1068.666,-57.944,439.348,172.387,23.692,154.328
C06852=1068.673,-57.695,439.336,172.388,23.693,154.328
C06853=1068.679,-57.445,439.324,172.390,23.695,154.328
C06854=1068.685,-57.195,439.313,172.391,23.697,154.328
C06855=1068.691,-56.946,439.301,172.393,23.699,154.329
C06856=1068.697,-56.696,439.288,172.394,23.701,154.329
C06857=1068.704,-56.446,439.277,172.396,23.703,154.329
C06858=1068.710,-56.197,439.265,172.397,23.705,154.329
C06859=1068.716,-55.947,439.253,172.400,23.707,154.329
C06860=1068.722,-55.697,439.241,172.401,23.709,154.329
C06861=1068.728,-55.448,439.230,172.403,23.711,154.329
C06862=1068.734,-55.198,439.217,172.404,23.712,154.330
C06863=1068.741,-54.948,439.205,172.405,23.715,154.330
C06864=1068.747,-54.699,439.194,172.407,23.717,154.330
C06865=1068.752,-54.450,439.181,172.408,23.718,154.330
C06866=1068.759,-54.199,439.170,172.410,23.720,154.330
C06867=1068.765,-53.950,439.158,172.411,23.722,154.330
C06868=1068.771,-53.700,439.146,172.413,23.724,154.331
C06869=1068.777,-53.451,439.134,172.414,23.726,154.331
C06870=1068.783,-53.201,439.121,172.416,23.728,154.331
C06871=1068.790,-52.951,439.110,172.417,23.730,154.331
C06872=1068.796,-52.701,439.098,172.419,23.731,154.331
C06873=1068.802,-52.452,439.086,172.420,23.734,154.331
C06874=1068.808,-52.203,439.074,172.422,23.736,154.332
C06875=1068.815,-51.953,439.062,172.424,23.738,154.332
C06876=1068.821,-51.703,439.050,172.425,23.740,154.332
C06877=1068.827,-51.453,439.038,172.427,23.742,154.332
C06878=1068.832,-51.204,439.026,172.428,23.744,154.332
C06879=1068.839,-50.954,439.014,172.430,23.745,154.332
C06880=1068.846,-50.705,439.002,172.431,23.747,154.332
C06881=1068.852,-50.455,438.990,172.433,23.750,154.333
C06882=1068.859,-50.178,438.976,172.434,23.752,154.333
C06883=1068.865,-49.901,438.963,172.436,23.754,154.333
C06884=1068.871,-49.624,438.949,172.438,23.756,154.333
C06885=1068.879,-49.346,438.936,172.439,23.759,154.333
C06886=1068.884,-49.097,438.924,172.441,23.760,154.334
C06887=1068.890,-48.847,438.911,172.442,23.763,154.334
C06888=1068.897,-48.597,438.899,172.444,23.765,154.334
C06889=1068.902,-48.348,438.887,172.445,23.767,154.334
C06890=1068.908,-48.098,438.875,172.446,23.769,154.334
C06891=1068.914,-47.849,438.863,172.448,23.771,154.335
C06892=1068.920,-47.599,438.850,172.450,23.773,154.335
C06893=1068.926,-47.349,438.837,172.452,23.775,154.335
C06894=1068.933,-47.099,438.826,172.453,23.777,154.335
C06895=1068.938,-46.850,438.813,172.455,23.779,154.335
C06896=1068.944,-46.600,438.801,172.456,23.782,154.336
C06897=1068.950,-46.350,438.788,172.457,23.783,154.336
C06898=1068.957,-46.101,438.776,172.459,23.785,154.336
C06899=1068.962,-45.852,438.764,172.460,23.788,154.336
C06900=1068.968,-45.602,438.752,172.462,23.790,154.336
C06901=1068.975,-45.352,438.740,172.463,23.791,154.336
C06902=1068.980,-45.102,438.727,172.465,23.794,154.337
C06903=1068.987,-44.853,438.714,172.466,23.796,154.337
C06904=1068.993,-44.604,438.702,172.467,23.798,154.337
C06905=1068.999,-44.354,438.690,172.469,23.800,154.337
C06906=1069.005,-44.104,438.677,172.470,23.802,154.337
C06907=1069.010,-43.855,438.664,172.472,23.804,154.338
C06908=1069.017,-43.605,438.653,172.474,23.806,154.338
C06909=1069.023,-43.355,438.640,172.476,23.809,154.338
C06910=1069.029,-43.105,438.627,172.477,23.811,154.338
C06911=1069.034,-42.856,438.615,172.478,23.813,154.338
C06912=1069.041,-42.607,438.603,172.480,23.815,154.339
C06913=1069.047,-42.357,438.590,172.481,23.817,154.339
C06914=1069.053,-42.107,438.577,172.483,23.819,154.339
C06915=1069.060,-41.858,438.565,172.484,23.821,154.339
C06916=1069.066,-41.608,438.553,172.485,23.824,154.339
C06917=1069.071,-41.358,438.540,172.487,23.825,154.340
C06918=1069.078,-41.109,438.527,172.488,23.827,154.340
C06919=1069.084,-40.860,438.516,172.490,23.830,154.340
C06920=1069.090,-40.610,438.503,172.491,23.831,154.340
C06921=1069.095,-40.360,438.490,172.493,23.834,154.340
C06922=1069.101,-40.110,438.478,172.494,23.836,154.341
C06923=1069.108,-39.861,438.465,172.496,23.839,154.341
C06924=1069.114,-39.611,438.453,172.498,23.840,154.341
C06925=1069.120,-39.362,438.440,172.499,23.842,154.341
C06926=1069.126,-39.112,438.428,172.501,23.845,154.341
C06927=1069.132,-38.862,438.414,172.502,23.846,154.342
C06928=1069.139,-38.613,438.402,172.504,23.849,154.342
C06929=1069.145,-38.363,438.390,172.505,23.851,154.342
C06930=1069.150,-38.114,438.378,172.506,23.853,154.342
C06931=1069.156,-37.864,438.364,172.508,23.856,154.342
C06932=1069.162,-37.615,438.352,172.509,23.857,154.343
C06933=1069.168,-37.365,438.339,172.511,23.860,154.343
C06934=1069.174,-37.115,438.326,172.512,23.862,154.343
C06935=1069.180,-36.866,438.313,172.513,23.864,154.343
C06936=1069.186,-36.616,438.301,172.515,23.866,154.343
C06937=1069.192,-36.366,438.288,172.516,23.868,154.344
C06938=1069.198,-36.117,438.275,172.518,23.871,154.344
C06939=1069.204,-35.867,438.262,172.520,23.873,154.344
C06940=1069.210,-35.617,438.249,172.521,23.875,154.344
C06941=1069.216,-35.368,438.237,172.523,23.877,154.345
C06942=1069.222,-35.118,438.224,172.524,23.880,154.345
C06943=1069.228,-34.869,438.211,172.525,23.882,154.345
C06944=1069.234,-34.619,438.199,172.527,23.884,154.345
C06945=1069.240,-34.369,438.186,172.528,23.886,154.346
C06946=1069.246,-34.093,438.172,172.530,23.889,154.346
C06947=1069.254,-33.816,438.157,172.532,23.892,154.346
C06948=1069.260,-33.539,438.143,172.533,23.894,154.346
C06949=1069.266,-33.262,438.128,172.535,23.896,154.346
C06950=1069.272,-33.013,438.116,172.536,23.898,154.347
C06951=1069.279,-32.763,438.103,172.537,23.901,154.347
C06952=1069.285,-32.513,438.090,172.539,23.902,154.347
C06953=1069.291,-32.264,438.077,172.540,23.905,154.347
C06954=1069.297,-32.014,438.064,172.542,23.907,154.348
C06955=1069.303,-31.764,438.052,172.544,23.909,154.348
C06956=1069.309,-31.515,438.038,172.545,23.912,154.348
C06957=1069.315,-31.265,438.026,172.547,23.914,154.348
C06958=1069.321,-31.016,438.012,172.548,23.916,154.348
C06959=1069.327,-30.766,438.000,172.549,23.919,154.349
C06960=1069.333,-30.517,437.987,172.551,23.920,154.349
C06961=1069.339,-30.267,437.974,172.552,23.923,154.349
C06962=1069.345,-30.018,437.961,172.554,23.925,154.349
C06963=1069.351,-29.768,437.948,172.555,23.927,154.350
C06964=1069.357,-29.519,437.935,172.556,23.929,154.350
C06965=1069.363,-29.269,437.922,172.558,23.932,154.350
C06966=1069.369,-29.019,437.909,172.559,23.934,154.350
C06967=1069.376,-28.770,437.896,172.561,23.936,154.351
C06968=1069.381,-28.520,437.883,172.562,23.938,154.351
C06969=1069.388,-28.271,437.870,172.563,23.940,154.351
C06970=1069.394,-28.021,437.858,172.566,23.943,154.351
C06971=1069.400,-27.772,437.844,172.567,23.946,154.351
C06972=1069.407,-27.522,437.831,172.569,23.947,154.352
C06973=1069.413,-27.272,437.818,172.570,23.950,154.352
C06974=1069.419,-27.023,437.805,172.571,23.952,154.352
C06975=1069.424,-26.773,437.792,172.573,23.954,154.352
C06976=1069.430,-26.523,437.778,172.574,23.956,154.353
C06977=1069.436,-26.274,437.765,172.575,23.959,154.353
C06978=1069.442,-26.024,437.753,172.577,23.961,154.353
C06979=1069.448,-25.775,437.739,172.578,23.964,154.353
C06980=1069.454,-25.525,437.725,172.580,23.965,154.354
C06981=1069.460,-25.275,437.713,172.581,23.968,154.354
C06982=1069.466,-25.026,437.700,172.582,23.970,154.354
C06983=1069.472,-24.777,437.686,172.584,23.973,154.354
C06984=1069.477,-24.527,437.673,172.585,23.975,154.355
C06985=1069.484,-24.277,437.660,172.587,23.978,154.355
C06986=1069.490,-24.028,437.647,172.589,23.980,154.355
C06987=1069.495,-23.778,437.634,172.590,23.982,154.355
C06988=1069.501,-23.529,437.620,172.591,23.985,154.356
C06989=1069.508,-23.279,437.607,172.593,23.987,154.356
C06990=1069.514,-23.029,437.593,172.594,23.989,154.356
C06991=1069.519,-22.779,437.580,172.596,23.991,154.356
C06992=1069.526,-22.530,437.567,172.597,23.994,154.357
C06993=1069.532,-22.281,437.554,172.598,23.996,154.357
C06994=1069.537,-22.031,437.540,172.600,23.998,154.357
C06995=1069.543,-21.781,437.527,172.601,24.001,154.357
C06996=1069.550,-21.532,437.514,172.602,24.003,154.358
C06997=1069.555,-21.282,437.500,172.604,24.005,154.358
C06998=1069.562,-21.032,437.486,172.605,24.007,154.358
C06999=1069.568,-20.783,437.473,172.607,24.010,154.358
C07000=1069.573,-20.533,437.460,172.608,24.012,154.359
C07001=1069.579,-20.284,437.447,172.610,24.015,154.359
C07002=1069.586,-20.034,437.434,172.612,24.017,154.359
C07003=1069.591,-19.785,437.420,172.613,24.020,154.359
C07004=1069.597,-19.536,437.406,172.614,24.022,154.360
C07005=1069.604,-19.286,437.393,172.616,24.024,154.360
C07006=1069.610,-19.036,437.379,172.617,24.026,154.360
C07007=1069.616,-18.786,437.366,172.618,24.029,154.360
C07008=1069.622,-18.537,437.353,172.620,24.031,154.361
C07009=1069.627,-18.287,437.339,172.621,24.034,154.361
C07010=1069.634,-18.010,437.324,172.622,24.036,154.361
C07011=1069.641,-17.732,437.310,172.625,24.039,154.361
C07012=1069.648,-17.455,437.295,172.626,24.041,154.362
C07013=1069.654,-17.178,437.279,172.627,24.044,154.362
C07014=1069.661,-16.928,437.266,172.629,24.046,154.362
C07015=1069.667,-16.678,437.252,172.630,24.048,154.363
C07016=1069.672,-16.428,437.239,172.631,24.051,154.363
C07017=1069.679,-16.179,437.226,172.634,24.054,154.363
C07018=1069.685,-15.929,437.212,172.635,24.056,154.363
C07019=1069.691,-15.680,437.198,172.636,24.058,154.364
C07020=1069.697,-15.430,437.185,172.638,24.061,154.364
C07021=1069.703,-15.181,437.171,172.639,24.063,154.364
C07022=1069.709,-14.931,437.158,172.641,24.065,154.364
C07023=1069.715,-14.681,437.144,172.642,24.067,154.365
C07024=1069.721,-14.432,437.130,172.643,24.070,154.365
C07025=1069.727,-14.182,437.117,172.645,24.072,154.365
C07026=1069.733,-13.933,437.103,172.646,24.075,154.365
C07027=1069.738,-13.683,437.089,172.647,24.077,154.366
C07028=1069.745,-13.434,437.076,172.649,24.079,154.366
C07029=1069.751,-13.184,437.062,172.650,24.082,154.366
C07030=1069.756,-12.934,437.048,172.651,24.084,154.367
C07031=1069.762,-12.685,437.035,172.653,24.087,154.367
C07032=1069.768,-12.436,437.021,172.654,24.089,154.367
C07033=1069.775,-12.186,437.007,172.656,24.092,154.367
C07034=1069.780,-11.937,436.993,172.658,24.094,154.368
C07035=1069.787,-11.687,436.979,172.659,24.096,154.368
C07036=1069.792,-11.438,436.966,172.660,24.099,154.368
C07037=1069.798,-11.187,436.951,172.662,24.101,154.368
C07038=1069.804,-10.938,436.938,172.663,24.104,154.369
C07039=1069.810,-10.689,436.924,172.664,24.106,154.369
C07040=1069.816,-10.439,436.911,172.666,24.108,154.369
C07041=1069.822,-10.189,436.897,172.667,24.111,154.370
C07042=1069.828,-9.940,436.882,172.669,24.113,154.370
C07043=1069.834,-9.691,436.869,172.670,24.116,154.370
C07044=1069.840,-9.441,436.855,172.671,24.118,154.370
C07045=1069.846,-9.191,436.841,172.673,24.120,154.371
C07046=1069.852,-8.942,436.828,172.674,24.123,154.371
C07047=1069.857,-8.692,436.814,172.675,24.126,154.371
C07048=1069.865,-8.443,436.799,172.677,24.129,154.372
C07049=1069.870,-8.193,436.785,172.679,24.131,154.372
C07050=1069.876,-7.944,436.772,172.680,24.133,154.372
C07051=1069.882,-7.694,436.758,172.681,24.136,154.372
C07052=1069.888,-7.444,436.744,172.683,24.138,154.373
C07053=1069.894,-7.196,436.730,172.684,24.140,154.373
C07054=1069.900,-6.946,436.716,172.686,24.143,154.373
C07055=1069.907,-6.696,436.703,172.687,24.145,154.373
C07056=1069.912,-6.446,436.689,172.688,24.148,154.374
C07057=1069.918,-6.197,436.674,172.690,24.150,154.374
C07058=1069.925,-5.947,436.661,172.691,24.152,154.374
C07059=1069.930,-5.698,436.647,172.692,24.155,154.375
C07060=1069.936,-5.448,436.632,172.694,24.157,154.375
C07061=1069.943,-5.199,436.618,172.695,24.160,154.375
C07062=1069.948,-4.949,436.605,172.696,24.162,154.375
C07063=1069.954,-4.699,436.590,172.698,24.164,154.376
C07064=1069.961,-4.450,436.576,172.700,24.167,154.376
C07065=1069.966,-4.201,436.563,172.701,24.170,154.376
C07066=1069.972,-3.951,436.548,172.703,24.172,154.376
C07067=1069.979,-3.701,436.535,172.704,24.174,154.377
C07068=1069.984,-3.452,436.520,172.705,24.177,154.377
C07069=1069.990,-3.202,436.506,172.707,24.179,154.377
C07070=1069.996,-2.953,436.492,172.708,24.182,154.378
C07071=1070.002,-2.704,436.478,172.709,24.184,154.378
C07072=1070.009,-2.454,436.464,172.711,24.187,154.378
C07073=1070.014,-2.205,436.450,172.712,24.189,154.379
C07074=1070.021,-1.925,436.433,172.713,24.192,154.379
C07075=1070.027,-1.646,436.418,172.716,24.195,154.379
C07076=1070.034,-1.367,436.403,172.717,24.198,154.380
C07077=1070.041,-1.088,436.386,172.718,24.200,154.380
C07078=1070.046,-0.838,436.372,172.719,24.203,154.380
C07079=1070.052,-0.588,436.358,172.721,24.206,154.381
C07080=1070.058,-0.339,436.343,172.722,24.208,154.381
C07081=1070.063,-0.090,436.329,172.724,24.211,154.381
C07082=1070.070,0.160,436.314,172.726,24.213,154.381
C07083=1070.075,0.410,436.300,172.727,24.216,154.382
C07084=1070.081,0.659,436.286,172.728,24.218,154.382
C07085=1070.087,0.909,436.272,172.730,24.221,154.382
C07086=1070.093,1.158,436.257,172.731,24.223,154.383
C07087=1070.099,1.408,436.243,172.732,24.226,154.383
C07088=1070.106,1.657,436.229,172.734,24.229,154.383
C07089=1070.111,1.906,436.215,172.735,24.231,154.383
C07090=1070.117,2.156,436.200,172.736,24.233,154.384
C07091=1070.123,2.406,436.186,172.738,24.236,154.384
C07092=1070.129,2.655,436.171,172.739,24.238,154.384
C07093=1070.135,2.905,436.157,172.740,24.241,154.385
C07094=1070.141,3.154,436.143,172.742,24.243,154.385
C07095=1070.147,3.404,436.129,172.743,24.246,154.385
C07096=1070.152,3.653,436.114,172.744,24.248,154.386
C07097=1070.158,3.903,436.100,172.746,24.252,154.386
C07098=1070.164,4.152,436.085,172.748,24.254,154.386
C07099=1070.171,4.402,436.070,172.749,24.256,154.386
C07100=1070.176,4.651,436.056,172.750,24.259,154.387
C07101=1070.182,4.900,436.042,172.752,24.261,154.387
C07102=1070.188,5.151,436.028,172.753,24.264,154.387
C07103=1070.194,5.400,436.013,172.754,24.266,154.388
C07104=1070.200,5.649,435.998,172.756,24.269,154.388
C07105=1070.206,5.899,435.984,172.757,24.271,154.388
C07106=1070.212,6.149,435.969,172.759,24.274,154.389
C07107=1070.218,6.397,435.955,172.760,24.276,154.389
C07108=1070.224,6.648,435.940,172.761,24.279,154.389
C07109=1070.230,6.897,435.926,172.762,24.281,154.390
C07110=1070.236,7.147,435.912,172.764,24.284,154.390
C07111=1070.242,7.396,435.897,172.765,24.286,154.390
C07112=1070.248,7.646,435.882,172.766,24.289,154.390
C07113=1070.254,7.895,435.867,172.769,24.292,154.391
C07114=1070.260,8.145,435.853,172.770,24.294,154.391
C07115=1070.266,8.394,435.839,172.771,24.296,154.391
C07116=1070.272,8.643,435.824,172.773,24.299,154.392
C07117=1070.277,8.893,435.810,172.774,24.302,154.392
C07118=1070.284,9.143,435.795,172.775,24.304,154.392
C07119=1070.290,9.392,435.780,172.777,24.307,154.392
C07120=1070.296,9.641,435.765,172.778,24.309,154.393
C07121=1070.302,9.892,435.751,172.779,24.312,154.393
C07122=1070.308,10.141,435.737,172.781,24.314,154.393
C07123=1070.314,10.390,435.722,172.782,24.317,154.394
C07124=1070.320,10.639,435.707,172.783,24.319,154.394
C07125=1070.326,10.889,435.693,172.785,24.321,154.394
C07126=1070.332,11.138,435.678,172.786,24.324,154.395
C07127=1070.338,11.388,435.663,172.787,24.327,154.395
C07128=1070.344,11.637,435.649,172.789,24.329,154.395
C07129=1070.350,11.887,435.634,172.791,24.332,154.395
C07130=1070.356,12.137,435.620,172.792,24.335,154.396
C07131=1070.362,12.386,435.604,172.794,24.337,154.396
C07132=1070.368,12.636,435.589,172.795,24.340,154.396
C07133=1070.374,12.885,435.575,172.796,24.342,154.397
C07134=1070.380,13.134,435.560,172.798,24.344,154.397
C07135=1070.386,13.384,435.545,172.799,24.347,154.397
C07136=1070.392,13.634,435.531,172.800,24.350,154.398
C07137=1070.398,13.883,435.516,172.802,24.352,154.398
C07138=1070.405,14.164,435.499,172.803,24.355,154.398
C07139=1070.412,14.445,435.483,172.805,24.358,154.399
C07140=1070.419,14.727,435.466,172.806,24.361,154.399
C07141=1070.425,15.008,435.449,172.808,24.364,154.399
C07142=1070.431,15.256,435.434,172.809,24.366,154.400
C07143=1070.437,15.506,435.419,172.810,24.368,154.400
C07144=1070.443,15.756,435.404,172.812,24.371,154.400
C07145=1070.449,16.005,435.389,172.814,24.374,154.401
C07146=1070.455,16.255,435.374,172.815,24.376,154.401
C07147=1070.461,16.504,435.360,172.816,24.379,154.401
C07148=1070.466,16.754,435.345,172.818,24.382,154.402
C07149=1070.473,17.004,435.330,172.819,24.384,154.402
C07150=1070.479,17.253,435.315,172.820,24.387,154.402
C07151=1070.484,17.503,435.300,172.822,24.389,154.403
C07152=1070.490,17.752,435.285,172.823,24.392,154.403
C07153=1070.496,18.001,435.270,172.824,24.395,154.403
C07154=1070.503,18.251,435.255,172.826,24.397,154.403
C07155=1070.508,18.500,435.240,172.827,24.399,154.404
C07156=1070.514,18.750,435.225,172.828,24.402,154.404
C07157=1070.521,18.999,435.210,172.830,24.405,154.404
C07158=1070.526,19.248,435.194,172.831,24.407,154.405
C07159=1070.532,19.498,435.179,172.832,24.410,154.405
C07160=1070.539,19.748,435.164,172.835,24.413,154.405
C07161=1070.544,19.997,435.149,172.836,24.415,154.406
C07162=1070.550,20.247,435.134,172.837,24.418,154.406
C07163=1070.556,20.496,435.119,172.839,24.420,154.406
C07164=1070.562,20.746,435.104,172.840,24.423,154.407
C07165=1070.568,20.995,435.089,172.841,24.426,154.407
C07166=1070.574,21.245,435.074,172.843,24.428,154.407
C07167=1070.579,21.494,435.059,172.844,24.430,154.408
C07168=1070.586,21.744,435.044,172.845,24.433,154.408
C07169=1070.592,21.993,435.028,172.847,24.436,154.408
C07170=1070.597,22.242,435.013,172.848,24.439,154.409
C07171=1070.603,22.492,434.998,172.849,24.441,154.409
C07172=1070.609,22.742,434.983,172.850,24.443,154.409
C07173=1070.615,22.991,434.968,172.852,24.446,154.410
C07174=1070.621,23.241,434.953,172.853,24.449,154.410
C07175=1070.628,23.490,434.937,172.854,24.451,154.410
C07176=1070.633,23.739,434.922,172.857,24.454,154.411
C07177=1070.639,23.989,434.907,172.858,24.457,154.411
C07178=1070.645,24.239,434.891,172.859,24.460,154.411
C07179=1070.650,24.487,434.877,172.861,24.462,154.411
C07180=1070.656,24.737,434.861,172.862,24.464,154.412
C07181=1070.663,24.986,434.846,172.863,24.467,154.412
C07182=1070.668,25.236,434.830,172.865,24.470,154.412
C07183=1070.674,25.485,434.816,172.866,24.472,154.413
C07184=1070.680,25.735,434.800,172.867,24.475,154.413
C07185=1070.687,25.984,434.784,172.869,24.477,154.413
C07186=1070.692,26.233,434.770,172.870,24.480,154.414
C07187=1070.698,26.483,434.754,172.871,24.483,154.414
C07188=1070.705,26.732,434.739,172.873,24.485,154.414
C07189=1070.710,26.982,434.723,172.874,24.488,154.415
C07190=1070.716,27.231,434.708,172.875,24.490,154.415
C07191=1070.722,27.481,434.693,172.877,24.493,154.415
C07192=1070.728,27.731,434.677,172.879,24.496,154.416
C07193=1070.734,27.980,434.662,172.880,24.498,154.416
C07194=1070.739,28.230,434.647,172.881,24.501,154.416
C07195=1070.746,28.479,434.631,172.883,24.504,154.417
C07196=1070.751,28.729,434.615,172.884,24.506,154.417
C07197=1070.758,28.978,434.600,172.885,24.509,154.417
C07198=1070.764,29.228,434.584,172.887,24.511,154.418
C07199=1070.769,29.477,434.569,172.888,24.514,154.418
C07200=1070.776,29.726,434.553,172.889,24.517,154.418
C07201=1070.781,29.976,434.538,172.891,24.520,154.419
C07202=1070.787,30.258,434.520,172.893,24.522,154.419
C07203=1070.795,30.541,434.503,172.894,24.525,154.419
C07204=1070.801,30.823,434.485,172.895,24.528,154.420
C07205=1070.808,31.106,434.468,172.897,24.531,154.420
C07206=1070.814,31.355,434.451,172.899,24.534,154.421
C07207=1070.819,31.604,434.437,172.900,24.537,154.421
C07208=1070.825,31.854,434.421,172.901,24.539,154.421
C07209=1070.831,32.104,434.405,172.903,24.542,154.421
C07210=1070.838,32.353,434.389,172.904,24.544,154.422
C07211=1070.843,32.603,434.374,172.905,24.547,154.422
C07212=1070.849,32.851,434.358,172.907,24.550,154.422
C07213=1070.855,33.101,434.343,172.908,24.553,154.423
C07214=1070.861,33.350,434.327,172.909,24.555,154.423
C07215=1070.867,33.600,434.311,172.911,24.558,154.424
C07216=1070.873,33.849,434.296,172.912,24.560,154.424
C07217=1070.878,34.099,434.280,172.913,24.563,154.424
C07218=1070.884,34.348,434.264,172.915,24.566,154.424
C07219=1070.890,34.598,434.249,172.917,24.568,154.425
C07220=1070.897,34.847,434.233,172.918,24.571,154.425
C07221=1070.902,35.097,434.217,172.919,24.574,154.425
C07222=1070.908,35.346,434.201,172.921,24.576,154.426
C07223=1070.915,35.596,434.186,172.922,24.579,154.426
C07224=1070.920,35.845,434.170,172.923,24.581,154.426
C07225=1070.926,36.095,434.155,172.925,24.584,154.427
C07226=1070.932,36.344,434.139,172.926,24.586,154.427
C07227=1070.938,36.593,434.123,172.927,24.589,154.428
C07228=1070.944,36.843,434.107,172.929,24.592,154.428
C07229=1070.950,37.092,434.091,172.930,24.594,154.428
C07230=1070.956,37.342,434.076,172.931,24.597,154.428
C07231=1070.962,37.591,434.060,172.934,24.600,154.429
C07232=1070.968,37.840,434.044,172.935,24.603,154.429
C07233=1070.973,38.090,434.028,172.936,24.605,154.429
C07234=1070.979,38.339,434.012,172.938,24.608,154.430
C07235=1070.985,38.589,433.996,172.939,24.610,154.430
C07236=1070.991,38.839,433.980,172.940,24.613,154.430
C07237=1070.997,39.088,433.965,172.942,24.616,154.431
C07238=1071.003,39.337,433.948,172.943,24.618,154.431
C07239=1071.009,39.587,433.933,172.944,24.621,154.431
C07240=1071.014,39.836,433.917,172.945,24.624,154.432
C07241=1071.020,40.085,433.901,172.947,24.626,154.432
C07242=1071.026,40.334,433.885,172.948,24.629,154.433
C07243=1071.032,40.584,433.869,172.949,24.631,154.433
C07244=1071.038,40.834,433.853,172.952,24.635,154.433
C07245=1071.044,41.083,433.836,172.953,24.637,154.433
C07246=1071.049,41.333,433.821,172.954,24.640,154.434
C07247=1071.055,41.582,433.805,172.956,24.642,154.434
C07248=1071.061,41.832,433.788,172.957,24.645,154.435
C07249=1071.067,42.080,433.773,172.958,24.648,154.435
C07250=1071.073,42.329,433.757,172.960,24.650,154.435
C07251=1071.079,42.579,433.741,172.961,24.653,154.436
C07252=1071.085,42.829,433.725,172.962,24.656,154.436
C07253=1071.091,43.078,433.709,172.964,24.658,154.436
C07254=1071.097,43.327,433.693,172.965,24.660,154.436
C07255=1071.103,43.577,433.676,172.966,24.663,154.437
C07256=1071.108,43.827,433.661,172.968,24.666,154.437
C07257=1071.114,44.076,433.645,172.970,24.669,154.438
C07258=1071.120,44.325,433.628,172.971,24.672,154.438
C07259=1071.126,44.575,433.611,172.972,24.674,154.438
C07260=1071.132,44.824,433.595,172.974,24.677,154.439
C07261=1071.137,45.074,433.579,172.975,24.680,154.439
C07262=1071.143,45.323,433.564,172.976,24.682,154.439
C07263=1071.148,45.572,433.547,172.978,24.685,154.440
C07264=1071.154,45.822,433.531,172.979,24.688,154.440
C07265=1071.160,46.071,433.515,172.980,24.691,154.440
C07266=1071.167,46.354,433.496,172.982,24.694,154.441
C07267=1071.174,46.636,433.478,172.984,24.697,154.441
C07268=1071.180,46.918,433.460,172.985,24.700,154.442
C07269=1071.186,47.201,433.441,172.987,24.703,154.442
C07270=1071.192,47.450,433.424,172.988,24.705,154.442
C07271=1071.198,47.700,433.408,172.990,24.708,154.443
C07272=1071.204,47.949,433.392,172.991,24.711,154.443
C07273=1071.210,48.198,433.376,172.992,24.714,154.443
C07274=1071.215,48.448,433.359,172.994,24.716,154.444
C07275=1071.221,48.697,433.342,172.995,24.719,154.444
C07276=1071.227,48.947,433.326,172.996,24.722,154.444
C07277=1071.233,49.196,433.310,172.998,24.724,154.445
C07278=1071.239,49.446,433.294,172.999,24.727,154.445
C07279=1071.244,49.695,433.277,173.001,24.730,154.445
C07280=1071.250,49.945,433.261,173.002,24.733,154.446
C07281=1071.256,50.194,433.244,173.004,24.735,154.446
C07282=1071.262,50.443,433.228,173.005,24.738,154.446
C07283=1071.268,50.693,433.212,173.006,24.741,154.447
C07284=1071.273,50.942,433.195,173.008,24.743,154.447
C07285=1071.279,51.192,433.179,173.009,24.746,154.448
